// TIA Portal V16 program export: 4 tag tables, 2 data types, 7 data blocks, 42 code blocks (in call order from the OBs), 94 instance data blocks

VAR_GLOBAL   // PLC tag table "Default tag table"
   "Drive 1 Ready" AT %I0.0 : Bool;   // +MC-21K2:1 - Drive 1 Ready
   "Drive 2 Ready" AT %I0.1 : Bool;   // +MC-21K2:5 - Drive 2 Ready
   "Drive 3 Ready" AT %I0.2 : Bool;   // +MC-21K2:2 - Drive 3 Ready
   "Drive 4 Ready" AT %I0.3 : Bool;   // +MC-21K2:6 - Drive 4 Ready
   "Drive 5 Ready" AT %I0.4 : Bool;   // +MC-21K2:3 - Drive 5 Ready
   "Sensor Trechter" AT %I0.5 : Bool;   // +MC-21K2:7 - Sensor Trechter
   "Sensor Op Band" AT %I0.6 : Bool;   // +MC-21K2:4 Sensor Op Band
   "Sensor Wals (Option)" AT %I0.7 : Bool;   // +MC-21K2:8 - Sensor Wals (Option)
   "ESB Oke" AT %I1.0 : Bool;   // +MC-21K3:1 - ESB Oke
   "ESB Pressend" AT %I1.1 : Bool;   // +MC-21K3:5 - ESB Pressend
   "Reset Active" AT %I1.2 : Bool;   // +MC-21K3:2 - Reset Active
   "Noodsleutel(1)" AT %I1.3 : Bool;   // +MC-21K3:6 - NOODSLEUTEL
   "Alle uitgangen(1)" AT %I1.4 : Bool;   // +MC-21K3:3 - Alle uitgangen
   "Door 1 NC contact" AT %I1.5 : Bool;   // +MC-21K3:7 - Safety Doorswitch 1
   "Door 1 NO contact" AT %I1.6 : Bool;   // +MC-21K3:4 - Safety Doorswitch 1 Normaly open
   "Door 2 NC contact" AT %I1.7 : Bool;   // +MC-21K3:8 - Safety Doorswitch 2
   "Spare(5)" AT %I3.0 : Bool;
   "Spare(6)" AT %I3.1 : Bool;
   "Spare(10)" AT %I180.0 : Bool;   // Spare
   "Spare(11)" AT %I180.1 : Bool;   // Spare
   "Spare(12)" AT %I3.4 : Bool;   // Spare
   "Spare(13)" AT %I3.5 : Bool;   // Spare
   "Spare(14)" AT %I3.6 : Bool;   // Spare
   "Spare(15)" AT %I3.7 : Bool;   // Spare
   "Programma 1" AT %I2.0 : Bool;   // +MC-21K4:1 - Programma 1
   "Programma 2" AT %I2.1 : Bool;   // +MC-21K4:5 - Programma 2 (Option)
   "Programma 3" AT %I2.2 : Bool;   // +MC-21K4:2 - Programma 3
   Cleaning AT %I2.3 : Bool;   // +MC-21K4:6 - Cleaning
   "Start Machine" AT %I2.4 : Bool;   // +MC-21K4:3 - Start Machine
   "Stop Machine" AT %I2.5 : Bool;   // +MC-21K4:7 - Stop Machine
   "Spare(16)" AT %I2.6 : Bool;   // Spare
   Encoder_Z_Puls AT %I2.7 : Bool;   // Spare
   "Safety Relais" AT %Q0.0 : Bool;   // +MC-21K6:1 - Safety Relais
   "Bel Storing" AT %Q0.1 : Bool;   // +MC-21K6:5 - Bel Storing
   Spare AT %Q5.3 : Bool;   // Spare
   "Drive 1 RUN FWD" AT %Q1.0 : Bool;   // +MC-21K8:1 - Drive 1 RUN FWD
   "Drive 1 REV]" AT %Q1.1 : Bool;   // +MC-21K8:5 - Drive 1 REV
   "Drive 1 Speed 1" AT %Q1.2 : Bool;   // +MC-21K8:2 - Drive 1 Speed 1
   "Drive 1 Speed 2" AT %Q1.3 : Bool;   // +MC-21K8:6 - Drive 1 Speed 2
   "Spare(3)" AT %Q1.4 : Bool;   // Spare
   "Drive 2 RUN FWD" AT %Q1.5 : Bool;   // +MC-21K8:7 - Drive 2 RUN FWD
   "Drive 2 REV" AT %Q1.6 : Bool;   // +MC-21K8:4 - Drive 2 REV
   "Drive 2 Speed 1" AT %Q1.7 : Bool;   // +MC-21K8:8 - Drive 2 Speed 1
   "Drive 2 Speed 2" AT %Q2.0 : Bool;   // +MC-21K9:1 - Drive 2 Speed 2
   "Spare(4)" AT %Q2.1 : Bool;   // Spare
   "Drive 3 RUN FWD" AT %Q2.2 : Bool;   // +MC-21K9:2 - Drive 3 RUN FWD
   "Drive 3 REV" AT %Q2.3 : Bool;   // +MC-21K9:6 - Drive 3 REV
   "Drive 3 Speed 1" AT %Q2.4 : Bool;   // +MC-21K9:3 - Drive 3 Speed 1
   "Drive 3 Speed 2" AT %Q2.5 : Bool;   // +MC-21K9:7 - Drive 3 Speed 2
   "Spare(21)" AT %Q2.6 : Bool;   // Spare
   "Drive 4 RUN FWD" AT %Q2.7 : Bool;   // +MC-21K9:8 - Drive 4 RUN FWD
   "Drive 4 REV" AT %Q3.0 : Bool;   // +MC-21K10:1 - Drive 4 REV
   "Drive 4 Speed 1" AT %Q3.1 : Bool;   // +MC-21K10:5 - Drive 4 Speed 1
   "Drive 4 Speed 2" AT %Q3.2 : Bool;   // +MC-21K10:2 - Drive 4 Speed 2
   "Spare(22)" AT %Q3.3 : Bool;   // Spare
   "Drive 5 RUN FWD" AT %Q3.4 : Bool;   // +MC-21K10:3 - Drive 5 RUN FWD
   "Drive 5 REV" AT %Q3.5 : Bool;   // +MC-21K10:7 - Drive 5 REV
   "Drive 5 Speed 1" AT %Q3.6 : Bool;   // +MC-21K10:4 - Drive 5 Speed 1
   "Drive 5 Speed 2" AT %Q3.7 : Bool;   // +MC-21K10:8 - Drive 5 Speed 2
   "Spare(23)" AT %Q4.0 : Bool;   // Spare
   "LED Programma 1" AT %Q4.1 : Bool;   // +MC-21K11:5 - LED Programma 1
   "LED Programma 2" AT %Q4.2 : Bool;   // +MC-21K11:2 - LED Programma 2
   "LED Programma 3" AT %Q4.3 : Bool;   // +MC-21K11:6 - LED Programma 3
   "LED E-STOP" AT %Q0.2 : Bool;   // +MC-21K6:2- LED E-STOP
   "LED RUN" AT %Q4.5 : Bool;   // +MC-21K11:7 - LED RUN
   "Valve 1" AT %Q4.6 : Bool;   // +MC-21K11:4 - Valve 1
   "Valve 2" AT %Q4.7 : Bool;   // +MC-21K11:8 - Valve 2
   "Valve 3" AT %Q5.0 : Bool;   // +MC-21K12:1 - Valve 3
   "Valve 4" AT %Q5.1 : Bool;   // +MC-21K12:5 - Valve 4
   "Valve 5" AT %Q5.2 : Bool;   // +MC-21K12:2 - Valve 5
   Nootstopper AT %Q6.0 : Bool;   // Spare
   "Spare(2)" AT %Q6.1 : Bool;   // Spare
   "Spare(18)" AT %Q6.2 : Bool;   // Spare
   "Spare(19)" AT %Q6.3 : Bool;   // Spare
   "Spare(20)" AT %Q4.4 : Bool;   // Spare
   "Drive 1 Rapid Stop" AT %Q0.3 : Bool;   // +MC-21K6:6 - Drive 1 Rapid Stop
   "Drive 2 Rapid Stop" AT %Q0.4 : Bool;   // +MC-21K6:3 - Drive 2 Rapid Stop
   "Drive 3 Rapid Stop" AT %Q0.5 : Bool;   // +MC-21K6:7 - Drive 3 Rapid Stop
   "Drive 4 Rapid Stop" AT %Q0.6 : Bool;   // +MC-21K6:4 - Drive 4 Rapid Stop
   "Drive 5 Rapid Stop" AT %Q0.7 : Bool;   // +MC-21K6:8 - Drive 5 Rapid Stop
   "Systeem RUN" AT %M0.0 : Bool;   // Systeem RUN
   Tag_1 AT %M0.1 : Bool;
   Tag_2 AT %M0.2 : Bool;
   Tag_3 AT %M0.3 : Bool;
   Tag_4 AT %M0.4 : Bool;
   "Safety Feedback" AT %M0.6 : Bool;
   Tag_5 AT %M0.7 : Bool;
   Tag_6 AT %M1.0 : Bool;
   "ONC Drive 1 RUN FWD" AT %M10.0 : Bool;
   "ONC Drive 2 RUN FWD" AT %M10.1 : Bool;
   "ONC Drive 3 RUN FWD" AT %M10.2 : Bool;
   "ONC Drive 4 RUN FWD" AT %M10.3 : Bool;
   "ONC Drive 5 RUN FWD" AT %M10.4 : Bool;
   "ONC Drive 1 RUN FWD and Speed 1" AT %M10.5 : Bool;
   "ONC Drive 2 RUN FWD and Speed 1" AT %M10.6 : Bool;
   "ONC Drive 3 RUN FWD and Speed 1" AT %M10.7 : Bool;
   "ONC Drive 4 RUN FWD and Speed 1" AT %M11.0 : Bool;
   "ONC Drive 5 RUN FWD and Speed 1" AT %M11.1 : Bool;
   "ONC Drive 1 RUN FWD and Speed 2" AT %M11.2 : Bool;
   "ONC Drive 2 RUN FWD and Speed 2" AT %M11.3 : Bool;
   "ONC Drive 3 RUN FWD and Speed 2" AT %M11.4 : Bool;
   "ONC Drive 4 RUN FWD and Speed 2" AT %M11.5 : Bool;
   "ONC Drive 5 RUN FWD and Speed 2" AT %M11.6 : Bool;
   Startknop_Scherm AT %M15.0 : Bool;
   Stopknop_Scherm AT %M15.1 : Bool;
   Tag_7 AT %M110.1 : Bool;
   Reset_scherm AT %M15.2 : Bool;
   Sensor_op_band_memory AT %M15.3 : Bool;
   "System RUN_1" AT %M20.0 : Bool;
   ResetDelay AT %M20.1 : Bool;
   SensorWalsMemory AT %M20.2 : Bool;
   Timer_Memory AT %M20.3 : Bool;
   StopAll AT %M20.4 : Bool;
   Tag_8 AT %M100.3 : Bool;
   Tag_9 AT %M100.4 : Bool;
   Tag_10 AT %M0.5 : Bool;
   Tag_11 AT %M150.0 : Bool;
   Tag_12 AT %M101.1 : Bool;
   Tag_13 AT %T1 : Timer;
   Tag_14 AT %M300.0 : Bool;
   Tag_15 AT %M260.0 : Bool;
   Tag_16 AT %M300.1 : Bool;
   Tag_17 AT %M501.0 : Bool;
   Tag_18 AT %M500.1 : Bool;
   Tag_19 AT %M160.0 : Bool;
   Tag_20 AT %M150.5 : Bool;
   Tag_21 AT %QD256 : DWord;
   Tag_22 AT %QW260 : Word;
   Tag_23 AT %ID256 : DWord;
   Tag_24 AT %ID260 : DWord;
   Tag_25 AT %ID464 : DWord;
   Tag_26 AT %ID471 : DWord;
   Tag_27 AT %QW471 : Word;
   Tag_28 AT %QD464 : DWord;
   Tag_30 AT %IW205 : Int;
   SystemTime AT %MD2 : Time;
   Tag_31 AT %M5.0 : Bool;
   Lamp_Green AT %Q7.0 : Bool;
   Lamp_Blue AT %Q7.1 : Bool;
   Lamp_Yellow AT %Q7.2 : Bool;
   Lamp_Red AT %Q7.3 : Bool;
   Lamp_Buzzer AT %Q7.4 : Bool;
   PulseTimer AT %T0 : Timer;
   Zpuls_Encoder_Band_Set AT %M1.1 : Bool;
   Drive_1_RefRun AT %M1.2 : Bool;
   Tag_32 AT %QD110 : DWord;
   Tag_33 AT %QD111 : DWord;
   Tag_34 AT %QD112 : DWord;
   Tag_35 AT %QD113 : DWord;
   Tag_36 AT %QD114 : DWord;
   Tag_37 AT %QD115 : DWord;
   Tag_38 AT %QD116 : DWord;
   Tag_39 AT %QD117 : DWord;
   Tag_40 AT %QB110 : Byte;
   Tag_41 AT %QB111 : Byte;
   Tag_42 AT %QB112 : Byte;
   Tag_43 AT %QB113 : Byte;
   Tag_44 AT %IB110 : Byte;
   Tag_45 AT %IB111 : Byte;
   Tag_46 AT %IB112 : Byte;
   Tag_47 AT %IB113 : Byte;
   Tag_48 AT %IB114 : Byte;
   Tag_49 AT %IB115 : Byte;
   Tag_50 AT %IB116 : Byte;
   Tag_51 AT %IB117 : Byte;
   Tag_52 AT %QD260 : DWord;
   Tag_53 AT %QB114 : Byte;
   Tag_54 AT %QB115 : Byte;
   Tag_55 AT %QB116 : Byte;
   Tag_56 AT %QB117 : Byte;
   Tag_57 AT %QW256 : Word;
   Tag_58 AT %QW258 : Word;
   Tag_59 AT %IW256 : Word;
   Tag_60 AT %IW258 : Word;
   Tag_61 AT %QW112 : Word;
   "Blow Off Timed" AT %M1.3 : Bool;
   Stop_valve_6 AT %M1.4 : Bool;
   Valve_6_Manual AT %M1.5 : Bool;
   Valve_6_Auto AT %M1.6 : Bool;
END_VAR

VAR_GLOBAL   // PLC tag table "PositionControl"
   Counter1_IW100 AT %IW100 : Int;
   Counter2_IW102 AT %IW102 : Int;
   "Manual Jog Fwd" AT %M137.0 : Bool;
   "Manual Jog Rev" AT %M137.1 : Bool;
   ReferenceSwitchAxis3 AT %I3.0 : Bool;
   EncoderBand_Alive AT %IW110 : Int;
   EncoderBand_RawCounter AT %ID112 : DInt;
   EncoderBand_FineCounter AT %IW113 : Int;
   Zpuls_Encoder_Band AT %I110.3 : Bool;
   Enc1 AT %ID110 : DInt;
   Enc2 AT %ID111 : DInt;
   Enc3 AT %ID113 : DInt;
   "Zpuls_Encoder_Band(1)" AT %I113.3 : Bool;
   "Enc3(1)" AT %ID114 : DInt;
   "Enc3(2)" AT %ID115 : DInt;
   "Enc3(3)" AT %ID116 : DInt;
   "Enc3(4)" AT %ID117 : DInt;
   "Enc3(5)" AT %ID118 : DInt;
   "Enc3(6)" AT %IW112 : Int;
   Enable AT %QW110 : Word;
   MovePos2 AT %M222.0 : Bool;
   ActivateProductBufferV3 AT %M222.1 : Bool;
END_VAR

VAR_GLOBAL   // PLC tag table "Secund. Tags"
   Aanvoerband_Tag1 AT %M100.0 : Bool;
   Aanvoerband_Tag2 AT %M100.1 : Bool;
   Trechter_Bijvullen_Haltveroorzaker AT %M100.2 : Bool;
   Safety_Automatic AT %M100.5 : Bool;
   Safety_Override AT %M100.6 : Bool;
   RUN_Automatic AT %M100.7 : Bool;
   RUN_Manual AT %M101.0 : Bool;
   Invert_Trechter_Sensor AT %M101.2 : Bool;
   WalsSensorMemory AT %M101.3 : Bool;
   Disable_Module AT %M101.4 : Bool;
   Sensor_Trechter_Delayed AT %M101.5 : Bool;
   Positive_Flank AT %M101.6 : Bool;
   ProductSensor_Flank AT %M101.7 : Bool;
   ProductSensor_Rug AT %M102.0 : Bool;
   SensorRug AT %M102.1 : Bool;
   TimeCyclusEnd AT %M102.2 : Bool;
   CounterReset AT %M102.3 : Bool;
   StartTimer AT %M102.4 : Bool;
   StopTimer AT %M102.5 : Bool;
   SaveTimervalue AT %M102.6 : Bool;
   ResetTotalProducts AT %M102.7 : Bool;
   MaintenanceNeeded AT %M103.0 : Bool;
   RetainValues AT %M112.0 : Bool;
   "Retain_1_DontTouch!" AT %M112.1 : Bool;
   Safety_Doors AT %M112.2 : Bool;
   Overname_Linked_Drive1 AT %M112.3 : Bool;
   Drive_RefuseLinkingDrive1 AT %M112.4 : Bool;
   Drive_4_Speed1_Link AT %M112.5 : Bool;
   Drive_4_Speed1_Unlink AT %M112.6 : Bool;
   SafetyOK AT %M112.7 : Bool;
   Valve2_Pulse AT %M113.0 : Bool;
   TurnOffDrive2 AT %M113.1 : Bool;
   TurnOffDrive4 AT %M113.2 : Bool;
   TurnOff_InfeedTimeout AT %M113.3 : Bool;
END_VAR

VAR_GLOBAL   // PLC tag table "Tag table_1"
END_VAR

TYPE "ProductEntry"
// stored: IsFailsafeCompliant false
   STRUCT
      StartTime : Time := T#0ms;
      Active : Bool;
   END_STRUCT;
END_TYPE

TYPE "ProductTrack"
// stored: IsFailsafeCompliant false
   STRUCT
      StartPosition : DInt;
      Active : Bool;
   END_STRUCT;
END_TYPE

DATA_BLOCK "DB1"   // DB93
VERSION : 0.1
// stored: AutoNumber true, IsOnlyStoredInLoadMemory false, IsWriteProtectedInAS false
   VAR RETAIN
      DBB0 : DWord;
      DBB15 : DWord;
      DBB14 : DWord;
      DBB13 : DWord;
      DBB12 : DWord;
      DBB11 : DWord;
      DBB10 : DWord;
      DBB9 : DWord;
      DBB8 : DWord;
      DBB7 : DWord;
      DBB6 : DWord;
      DBB5 : DWord;
      DBB4 : DWord;
      DBB3 : DWord;
      DBB2 : DWord;
      DBB1 : DWord;
      DBD4 : DWord;
      DBD0 : DWord;
      "DBX4.0" : Bool;
   END_VAR
BEGIN
END_DATA_BLOCK

DATA_BLOCK "DB_EncoderBand"   // DB95
VERSION : 0.1
// stored: AutoNumber false, IsOnlyStoredInLoadMemory false, IsWriteProtectedInAS false
   VAR RETAIN
      ControlWord1 : DInt;
      ControlWord2 : DInt;
      FeedbackWord1 : DInt;
      FeedbackWord2 : DInt;
      EnableGate : Bool;
      ControlWord : Word;
      EncoderValue : DInt;
   END_VAR
BEGIN
END_DATA_BLOCK

DATA_BLOCK "Datablock_Encoder"   // DB96
VERSION : 0.1
// stored: AutoNumber true, IsOnlyStoredInLoadMemory false, IsWriteProtectedInAS false
BEGIN
END_DATA_BLOCK

DATA_BLOCK "PLCMemory"   // DB15
VERSION : 0.1
// stored: AutoNumber true, IsOnlyStoredInLoadMemory false, IsWriteProtectedInAS false
   VAR RETAIN
      Homing_Sensor_Wals_Offset_Test : Time := T#1S_200MS;   // Offset of homing position sensor wals
      Wals_Delay_Offset : Time := T#400MS;   // Offset of Wals on delay
      Safety_Delay : Time := T#5MS;   // Delay of safety high
      WalsCheck_Time : Time := T#5S;   // Time offset when wals slipping message is displayed
      ProductCheck_Time : Time := T#15S;   // Time offset when aanvoer not in position message is displayed
      ProductIntervalTime : Time := T#10s;   // Counts the time between 2 products
      ProductIntervalTime_1 : Time;   // Depends on ProductIntervalTimer
      ProductIntervalTime_2 : Time;   // Depends on ProductIntervalTimer_1
      TD_Products_Counter : Int;   // Counts the total amount of products with the Sensor Band
      UsernameMemory : String := 'Key';
      PasswordMemory : String := 'Key123';
      SpeedSettingsTakeover : Bool := True;   // Makes the speed of Overname the same as speed Drive 1
      SpeedSettingOvername : Bool;   // Parameter of setting the speed for Drive 4 (Overname)
      SpeedSettingBand : Bool;   // Parameter of setting the speed for Drive 1 (Band)
      TimingSettingOvername : Bool := True;   // Makes the timing of Overname the same as speed Drive 1
      EncoderPosition : Real;   // Real Value of Encoder Axis 3 (Wals)
      StepSize : Real := 0.0;   // Pulsfactor of Encoder Axis 3
      Desired_Encoder_Position : Real;
      Tolerance : Real := 0.0;
      "Encoder PulsOffset" : Time := T#3MS;
      Axis3_Ref_Pos : Real := 85.0;   // Refention position of Axis 3 without tolerance
      Reference_Position_Axis3 : Real;   // Refention position of Axis 3 with calculated tolerance
      ProductCount : Int;
      Axis3_ControlMode : Bool := true;
      Axis1_ControlMode : Bool := true;
      ProductsToProduce : Int;
      SystemTime : Time;
      Disable_Modules : Struct
         Disable_Band : Bool;
         Disable_Trilgoten : Bool;
         Disable_AanvoerWals : Bool;
         Disable_Aandruk1 : Bool;
         Disable_Aandruk2 : Bool;
         Disable_Aandruk3 : Bool;
         Disable_Blaaspuls : Bool;
         Disable_Retourband : Bool;
         Disable_Afsluiter : Bool;
         Disable_Nootstopper : Bool;
      END_STRUCT;
      Offset_Timers : Struct
         Trilgoten_Start_Offset : Time := T#10MS;   // Delay offset of start trilgoten
         Trilgoten_Stop_Offset : Time := T#10MS;   // Delay offset of stop trilgoten
         Aanvoer_Start_Offset : Time := T#10MS;   // Delay offset of start aanvoer
         Magazijn_Sensor_Delay : Time := T#15S;   // Delay on magazijn sensor.
         Aanvoer_Stop_Offset : Time := T#10MS;   // Delay offset of stop aanvoer
         Overname_Start_Offset : Time := T#5MS;   // Delay offset of start Overname
         Overname_Stop_Offset : Time := T#5MS;   // Delay offset of stop Overname
         Retourband_Start_Offset : Time := T#5ms;
         Retourband_Stop_Offset : Time := T#5ms;
         BlowOff_CycleTime : Time := T#500ms;
         Blow_Off_PulseTime : Time := T#500ms;
      END_STRUCT;
      ProductBuffer : Struct
         DelayTime : Time := T#7s;
         ProductsCount : Int;
         MoveTrigger : Bool;
         MoveFeedback : Bool;
         RestFeedback : Bool;
         InsertIndex : Int;
      END_STRUCT;
      ProductBufferBehindWals : Struct
         DelayTime : Time := T#1s_890MS;
         Product_Count : Int;
      END_STRUCT;
      ProductBufferNutStopper : Struct
         ProductCount : Int;
         TimeOpenNutstopper_PT : Time := T#200MS;
         TimeOpenNutstopper_ET : Time;
      END_STRUCT;
      ProductBuffer_1 : Struct
         DelayTime : Time := T#7s;
         ProductsCount : Int;
         MoveTrigger : Bool;
         MoveFeedback : Bool;
         RestFeedback : Bool;
         InsertIndex : Int;
      END_STRUCT;
      TriggerDistanceBand : DInt := 418000;
      TriggerDistanceAandruk : DInt := 500000;
      TriggerDistanceNutStopper : DInt := 459000;
      InfeedTimeOutPT : Time := T#2S;
      "Blow Off Timer on" : Time := T#2S;
      ResetManual : Bool;
      StartDevTestingInfeedSensor : Bool;
      SimulateSensor : Bool;
      PulsTimeBlowOff : Time := T#650ms;
      BlowOffPulse : Bool;
      OutputUserText : Struct
         Axis1 : Struct
            "User1.Text" : String := '(300) Manual Jogging';
            "User2.Text" : String := '(50) Automatic Production';
            "User3.Text" : String := '(1) Reference Run';
            "User4.Text" : String;
            CurrentUserText : String;
         END_STRUCT;
         Axis2 : Struct
            "User1.Text" : String := '(300) Manual Jogging';
            "User2.Text" : String := '(50) Automatic Production';
            "User3.Text" : String;
            "User4.Text" : String;
            CurrentUserText : String;
         END_STRUCT;
         Axis3 : Struct
            "User1.Text" : String := '(300) Manual Jogging Fwd';
            "User2.Text" : String := '(300) Manual Jogging Rev';
            "User3.Text" : String := '(50) Automatic Servomanager';
            "User4.Text" : String := '(1) Reference Run';
            CurrentUserText : String;
         END_STRUCT;
         Axis4 : Struct
            "User1.Text" : String := '(300) Manual Jogging';
            "User2.Text" : String := '(50) Automatic Production';
            "User3.Text" : String;
            "User4.Text" : String;
            CurrentUserText : String;
         END_STRUCT;
         Axis5 : Struct
            "User1.Text" : String := '(300) Manual Jogging';
            "User2.Text" : String := '(50) Automatic Production';
            "User3.Text" : String;
            "User4.Text" : String;
            CurrentUserText : String;
         END_STRUCT;
      END_STRUCT;
      Modules : Struct
         Valve_6 : "ModuleOutput";
         Valve_1 { S7_SetPoint := 'True'} : "ModuleOutput";
         Valve_3 { S7_SetPoint := 'True'} : "ModuleOutput";
         Valve_4 { S7_SetPoint := 'True'} : "ModuleOutput";
         Valve_5 { S7_SetPoint := 'True'} : "ModuleOutput";
      END_STRUCT;
   END_VAR
BEGIN
END_DATA_BLOCK

DATA_BLOCK "DB_SystemTimeCounter"   // DB68
VERSION : 0.1
// stored: AutoNumber true, IsOnlyStoredInLoadMemory false, IsWriteProtectedInAS false
   VAR RETAIN
      SystemTime : Time;
   END_VAR
BEGIN
END_DATA_BLOCK

DATA_BLOCK "Alarms"   // DB24
VERSION : 0.1
// stored: AutoNumber true, IsOnlyStoredInLoadMemory false, IsWriteProtectedInAS false
   VAR
      AlarmStruct : Struct
         Alarm_Product_Not_Position : Bool;
         Alarm_Axis_Not_Position : Bool;
         Alarm_Drive1 : Bool;
         Alarm_Drive2 : Bool;
         Alarm_Drive3 : Bool;
         Alarm_Drive4 : Bool;
         Alarm_Drive5 : Bool;
         "Alarm_To_Many_Products_Reset_Counter!" : Bool;
      END_STRUCT;
      AlarmsWord : Word;
      HMI_Alarm_Drive1 : Word;
      HMI_Alarm_Drive2 : Word;
      HMI_Alarm_Drive3 : Word;
      HMI_Alarm_Drive4 : Word;
      HMI_Alarm_Drive5 : Word;
   END_VAR
BEGIN
END_DATA_BLOCK

DATA_BLOCK "PositionManagement"   // DB51
VERSION : 0.1
// stored: AutoNumber true, IsOnlyStoredInLoadMemory false, IsWriteProtectedInAS false
   VAR RETAIN
      Data : Struct   // Data
         CntPlsPrev : DInt := 0;   // Flowpulsen vorige scan
         CntPlsDiff : DInt := 0;   // Flowpulsen verschil
         CntPlsAct : DInt := 0;   // Flowpulsen actueel
         DosActueel : Real := 0.0;   // Dosering actueel (not used)
         Actual_Axis3_Position : Real;   // Actual Position of Axis 3 stored in this datablock
         Actual_Axis1_Position : Real;
      END_STRUCT;
      "Axis 3" : Struct
         Values : Struct
            AxisName : String := 'Drive 3 - Wals';
            "Reference Position" : Int := 0;
            "Set Position" : Real := -50.0;
            "Rest Position" : Real := -25.0;
            Acceleration : Real := 0.0;
            Deacceleration : Real;
            "Axis Correction" : Real := 1.0E-06;
            "Position Offset" : Real := 35.0;
            Pulsfactor : Real := 0.82;
            Axis_Speed : Int := 0;
            ModuloFactor : Real := 360.0;
         END_STRUCT;
         Commands : Struct
            "Go To Rest" : Bool;
            "Start Ref Run" : Bool;
            "Take Over Pos" : Bool;
            "Go To Position" : Bool;
            "Jog Fwd" : Bool;
            "Jog Rev" : Bool;
            Axis_Brake : Bool;
            MasterWord : String;
            "Master Callback" : String;
         END_STRUCT;
         Messages : Struct
            "Axis Busy" : Bool;
            "Error Executing Command" : Bool;
            "Axis On Rest" : Bool;
            "Axis On Position" : Bool;
            "Drive State (Option)" : String;
            "Slip State" : String;
            AxisHasReference : Bool;
         END_STRUCT;
      END_STRUCT;
      Demo_Pos : Struct
         Desired_Pos : Real;
         Start : Bool;
         SetRefRunActive : Bool;
         RequestMove1 : Bool;
         RequestMove2 : Bool;
         PositionMove2 : Real := -50.0;
         PositionMove1 : Real := -250.0;
         Pos2Done : Bool;
         BrakeOnPos1 : Bool;
         BrakeOnPos2 : Bool;
         ManualSensorOverride : Bool;
      END_STRUCT;
      Axis_1 : Struct
         Values : Struct
            AxisName : String := 'Drive 1 - Infeed';
            "Reference Position" : Int := 0;
            "Set Position" : Real := 0.0;
            "Rest Position" : Real := 0.0;
            Acceleration : Real := 0.0;
            Deacceleration : Real;
            "Axis Correction" : Real := 1.0E-06;
            "Position Offset" : Real := 0.001;
            Pulsfactor : Real := -0.359;
            Axis_Speed : Int := 0;
            LimitEncValue : DInt := 0;
         END_STRUCT;
         Commands : Struct
            "Go To Rest" : Bool;
            "Start Ref Run" : Bool;
            "Take Over Pos" : Bool;
            "Go To Position" : Bool;
            "Jog Fwd" : Bool;
            "Jog Rev" : Bool;
            Axis_Brake : Bool;
            ReferenceSwitch : Bool;
            MasterWord : String;
            "Master Callback" : String;
         END_STRUCT;
         Messages : Struct
            "Axis Busy" : Bool;
            "Error Executing Command" : Bool;
            "Axis On Rest" : Bool;
            "Axis On Position" : Bool;
            "Drive State (Option)" : String;
            "Slip State" : String;
            AxisHasReferenceDelayed : Bool;
            AxisHasReference : Bool;
            SetAxisHasRefFromEnc : Bool;
            MaxOverflowValueDint : DInt := 16#8261A800;
         END_STRUCT;
      END_STRUCT;
   END_VAR
BEGIN
END_DATA_BLOCK

ORGANIZATION_BLOCK "OB1"   // OB1, LAD, ProgramCycle
TITLE = MAIN Program - Sweep
VERSION : 0.1
// MAIN Program Block (Release)
// stored: IsIECCheckEnabled false
   VAR_TEMP
      Temp_0 : Byte;
      Temp_1 : Byte;
      Temp_2 : Byte;
      Temp_3 : Byte;
      Temp_4 : Byte;
      Temp_5 : Byte;
      Temp_6 : Int;
      Temp_7 : Int;
      Temp_8 : Int;
      Temp_9 : Date_And_Time;
      Temp_10 : DWord;
      EncoderDirection : Bool;
      HomingActive : Bool;
      EncError : Bool;
      SafetyActive : Bool;
      "Spare Drive 6" : Bool;
      "Spare Drive 7" : Bool;
      "Spare Drive 8" : Bool;
      "Spare Drive 9" : Bool;
      "Spare Drive 10" : Bool;
      SAFE_OK_Signal : Bool;
      Raw_Position : Real;
      Encoder : Int;
      Gate : Bool;
      GATESTP : Bool;
      OTERRA : Bool;
      Direct : Bool;
      Prepar : Bool;
      CMPV1 : Bool;
      CMPV2 : Bool;
      RESSYNC : Bool;
      RESZERO : Bool;
      OTERR : Bool;
      UnscPos : Int;
      Sc_Pos : Int;
      ActEncPos : Real;
      Start_ReferenceRun : Bool;
      ReferenceSwitch_Input : Bool;
      "Reference Position" : Real;
      "Jog FWD" : Bool;
      "Jog REV" : Bool;
      RefSwitchTemp : Bool;
      RefPosDint : DInt;
      RefPosInt : Real;
      Start_Movement : Bool;
      ClockTime : Int;
      LT_Time : Date_And_Time;
      Summer : Bool;
      SystemStartUp : Bool;
      StartupLow : Bool;
      ManualSensorOverride : Bool;
      Axis1_ScaledPosition : Real;
      Axis1_ActualEncPosition : Real;
      ActivateProductBufferV2 : Bool;
      ActivateProductBufferV3 : Bool;
      SetZPulse : Bool;
      Enc2_AboveZero : DInt;
      MinValue : DInt;
      EncBelowZero : Bool;
      SafeEncValue : Real;
      Enc2_Real : Real;
      ScPos : Real;
      UseOldDriveManager : Bool;
      NotUsed : Bool;
      Door2 : Bool;
      Resettt : Bool;
      BlkMovReturn : Int;
      BlkMovReturn2 : Int;
      ServoAxis3RefRun : Bool;
   END_VAR
   VAR_TEMP   // added for the SCL form of the ladder/FBD networks
      _w1 : Bool;
   END_VAR
BEGIN

REGION Network 1: System Startup
   // Network for detecting System Start-up.
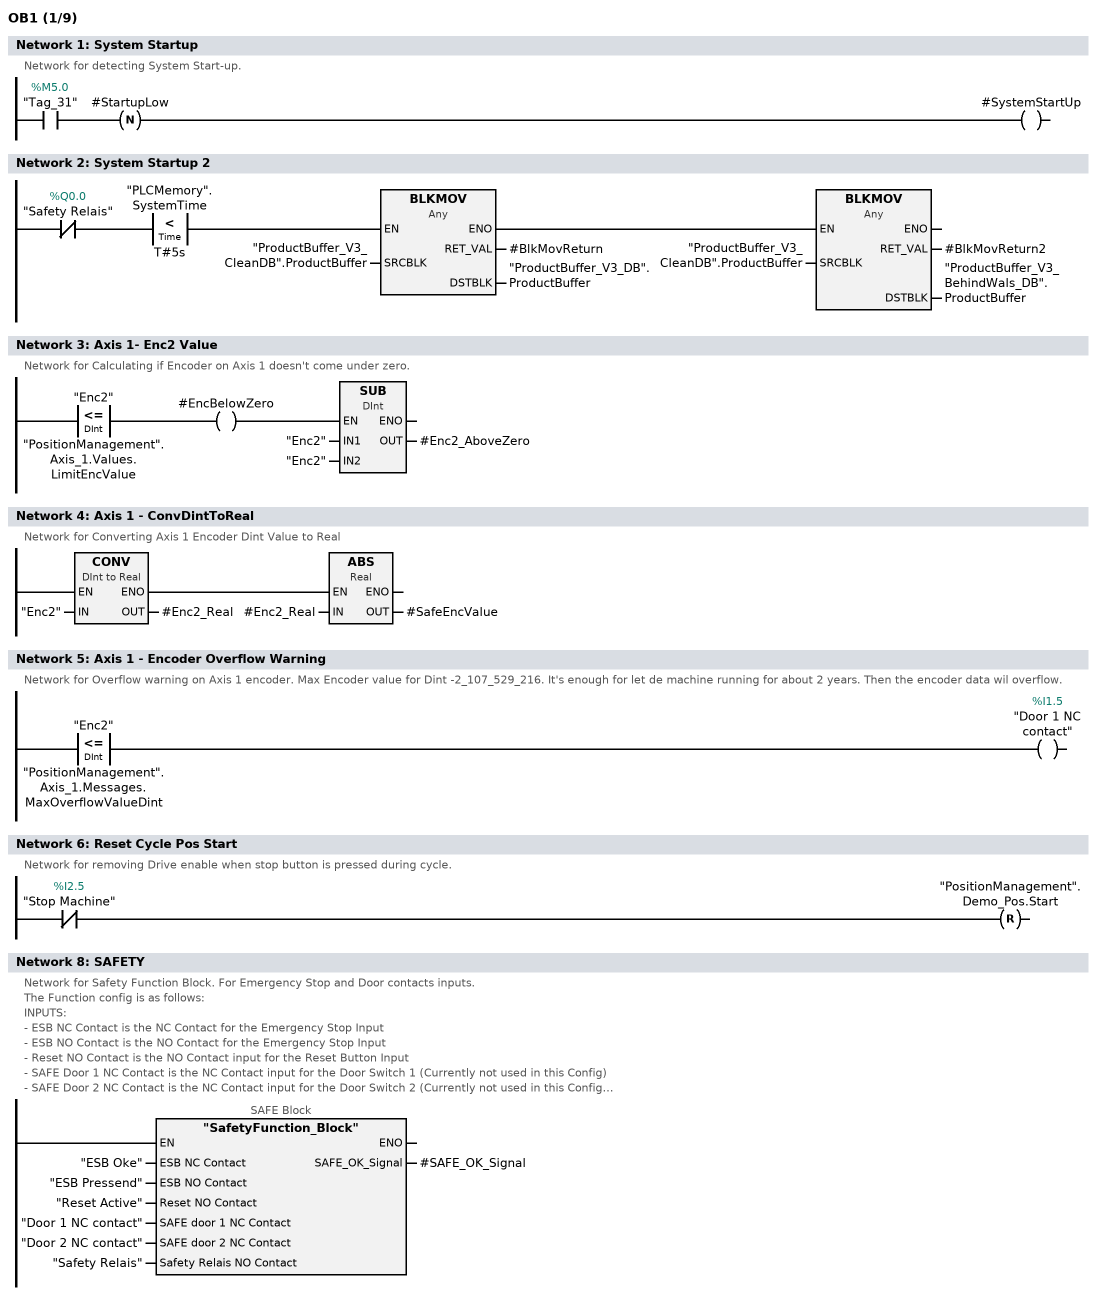
   RUNG wire#powerrail
      Contact( "Tag_31" )
      N_Trig( #StartupLow )
      Coil( #SystemStartUp )
   END_RUNG
   // the same network as SCL:
   #_w1 := NOT "Tag_31" AND #StartupLow;   // falling edge
   #StartupLow := "Tag_31";
   #SystemStartUp := #_w1;
END_REGION

REGION Network 2: System Startup 2
   RUNG wire#powerrail
      I_Contact( "Safety Relais" )
      { S7_Templates := "SrcType := Time" } LT_Contact(in1 := "PLCMemory".SystemTime, in2 := T#5s)
      { S7_Templates := "blk_type := Any" } BLKMOV(SRCBLK := "ProductBuffer_V3_CleanDB".ProductBuffer, RET_VAL => #BlkMovReturn, DSTBLK => "ProductBuffer_V3_DB".ProductBuffer)
      { S7_Templates := "blk_type := Any" } BLKMOV(SRCBLK := "ProductBuffer_V3_CleanDB".ProductBuffer, RET_VAL => #BlkMovReturn2, DSTBLK => "ProductBuffer_V3_BehindWals_DB".ProductBuffer)
   END_RUNG
   // the same network as SCL:
   #BlkMovReturn := BLKMOV(EN := NOT "Safety Relais" AND ("PLCMemory".SystemTime < T#5s),
                           SRCBLK := "ProductBuffer_V3_CleanDB".ProductBuffer,
                           DSTBLK => "ProductBuffer_V3_DB".ProductBuffer,
                           ENO => #_w1);
   IF #_w1 THEN
       #BlkMovReturn2 := BLKMOV(SRCBLK := "ProductBuffer_V3_CleanDB".ProductBuffer,
                               DSTBLK => "ProductBuffer_V3_BehindWals_DB".ProductBuffer);
   END_IF;
END_REGION

REGION Network 3: Axis 1- Enc2 Value
   // Network for Calculating if Encoder on Axis 1 doesn't come under zero.
   RUNG wire#powerrail
      { S7_Templates := "SrcType := DInt" } LE_Contact(in1 := "Enc2", in2 := "PositionManagement".Axis_1.Values.LimitEncValue)
      Coil( #EncBelowZero )
      { S7_Templates := "SrcType := DInt"; S7_GenerateENO := "TRUE" } Sub(in1 := "Enc2", in2 := "Enc2", out => #Enc2_AboveZero)
   END_RUNG
   // the same network as SCL:
   #EncBelowZero := "Enc2" <= "PositionManagement".Axis_1.Values.LimitEncValue;
   IF #EncBelowZero THEN #Enc2_AboveZero := "Enc2" - "Enc2"; END_IF;
END_REGION

REGION Network 4: Axis 1 - ConvDintToReal
   // Network for Converting Axis 1 Encoder Dint Value to Real
   RUNG wire#powerrail
      { S7_Templates := "[SrcType := DInt, DestType := Real]"; S7_GenerateENO := "TRUE" } Convert(in := "Enc2", out => #Enc2_Real)
      { S7_Templates := "SrcType := Real"; S7_GenerateENO := "TRUE" } Abs(in := #Enc2_Real, out => #SafeEncValue)
   END_RUNG
   // the same network as SCL:
   // ENO of a box is taken as its EN; it also drops when the box reports an error
   #Enc2_Real := DINT_TO_REAL("Enc2");
   #SafeEncValue := ABS(#Enc2_Real);
END_REGION

REGION Network 5: Axis 1 - Encoder Overflow Warning
   // Network for Overflow warning on Axis 1 encoder. Max Encoder value for Dint -2_107_529_216. It's enough for let de machine running for about 2 years. Then the encoder data wil overflow.
   RUNG wire#powerrail
      { S7_Templates := "SrcType := DInt" } LE_Contact(in1 := "Enc2", in2 := "PositionManagement".Axis_1.Messages.MaxOverflowValueDint)
      Coil( "Door 1 NC contact" )
   END_RUNG
   // the same network as SCL:
   "Door 1 NC contact" := "Enc2" <= "PositionManagement".Axis_1.Messages.MaxOverflowValueDint;
END_REGION

REGION Network 6: Reset Cycle Pos Start
   // Network for removing Drive enable when stop button is pressed during cycle.
   RUNG wire#powerrail
      I_Contact( "Stop Machine" )
      R_Coil( "PositionManagement".Demo_Pos.Start )
   END_RUNG
   // the same network as SCL:
   IF NOT "Stop Machine" THEN "PositionManagement".Demo_Pos.Start := FALSE; END_IF;
END_REGION

REGION Network 7: Retain Veriables (Not Used)
   // Spare Network Currently not used
END_REGION

REGION Network 8: SAFETY
   // Network for Safety Function Block. For Emergency Stop and Door contacts inputs.
   // The Function config is as follows:
   // 
   // INPUTS:
   // - ESB NC Contact is the NC Contact for the Emergency Stop Input
   // - ESB NO Contact is the NO Contact for the Emergency Stop Input
   // - Reset NO Contact is the NO Contact input for the Reset Button Input
   // - SAFE Door 1 NC Contact is the NC Contact input for the Door Switch 1 (Currently not used in this Config)
   // - SAFE Door 2 NC Contact is the NC Contact input for the Door Switch 2 (Currently not used in this Config)
   // - Safety Relais NO Contact is the NO Contact Input for feedback whenether the Safety Relais is powered or not.
   // 
   // OUTPUTS:
   // - SAFE_OK_Signal is the output for the SAFE OK signal, it's HIGH when all safety inputs are HIGH, en when Reset is given.
   RUNG wire#powerrail
      "SafetyFunction_Block"("ESB NC Contact" := "ESB Oke", "ESB NO Contact" := "ESB Pressend", "Reset NO Contact" := "Reset Active", "SAFE door 1 NC Contact" := "Door 1 NC contact", "SAFE door 2 NC Contact" := "Door 2 NC contact", "Safety Relais NO Contact" := "Safety Relais", SAFE_OK_Signal => #SAFE_OK_Signal)   // SAFE Block
   END_RUNG
   // the same network as SCL:
   "SafetyFunction_Block"("ESB NC Contact" := "ESB Oke",   // SAFE Block
                          "ESB NO Contact" := "ESB Pressend",
                          "Reset NO Contact" := "Reset Active",
                          "SAFE door 1 NC Contact" := "Door 1 NC contact",
                          "SAFE door 2 NC Contact" := "Door 2 NC contact",
                          "Safety Relais NO Contact" := "Safety Relais",
                          SAFE_OK_Signal => #SAFE_OK_Signal);
END_REGION

REGION Network 9: SAFE Signal
   // Network for internal SAFETY OK Confirmation
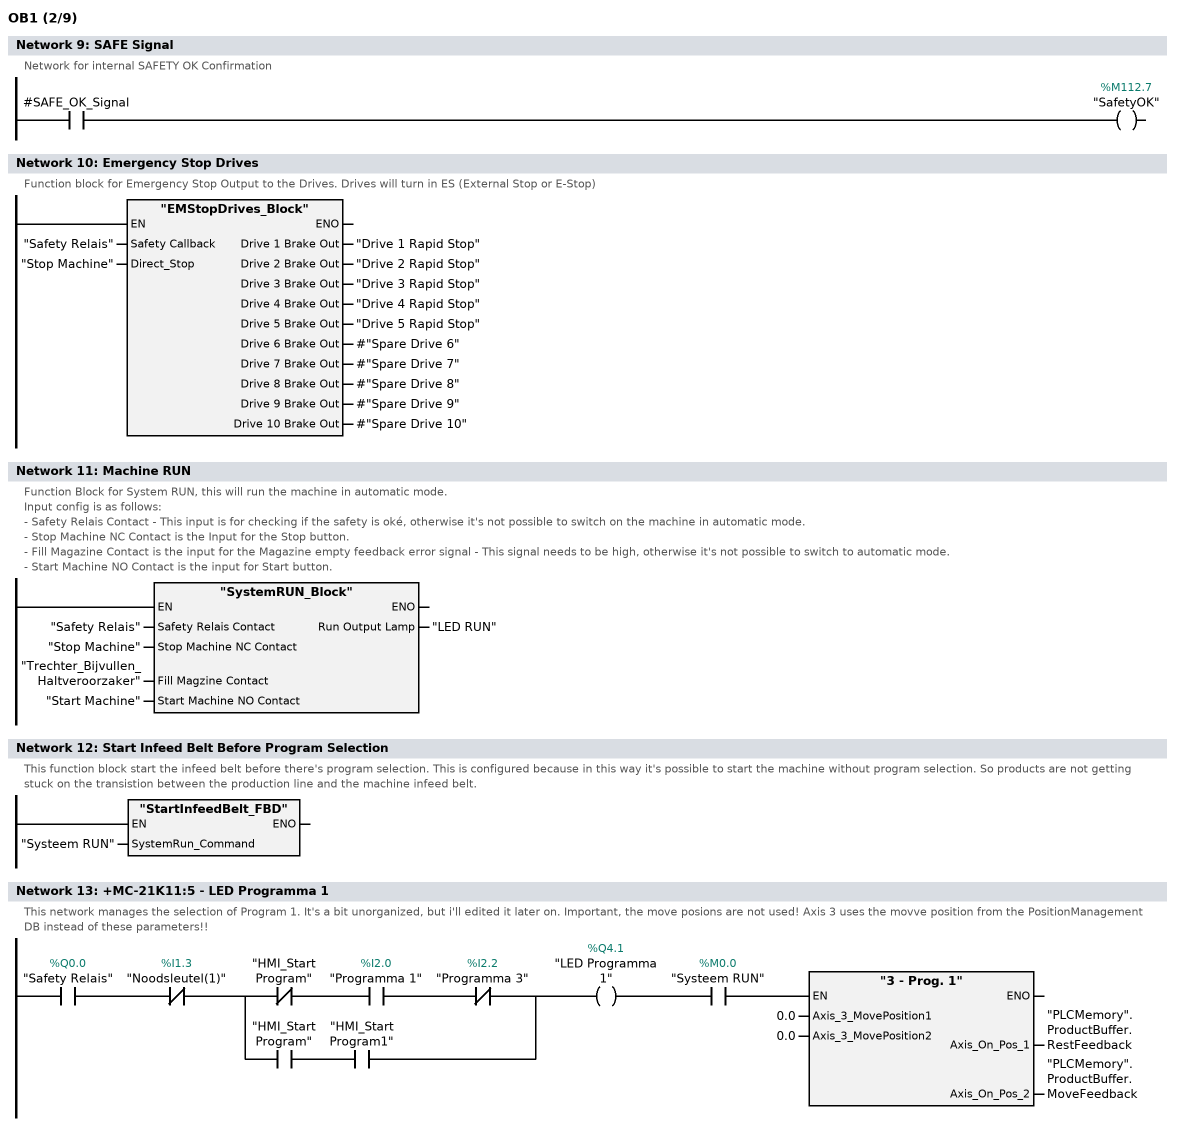
   RUNG wire#powerrail
      Contact( #SAFE_OK_Signal )
      Coil( "SafetyOK" )
   END_RUNG
   // the same network as SCL:
   "SafetyOK" := #SAFE_OK_Signal;
END_REGION

REGION Network 10: Emergency Stop Drives
   // Function block for Emergency Stop Output to the Drives. Drives will turn in ES (External Stop or E-Stop)
   RUNG wire#powerrail
      "EMStopDrives_Block"("Safety Callback" := "Safety Relais", Direct_Stop := "Stop Machine", "Drive 1 Brake Out" => "Drive 1 Rapid Stop", "Drive 2 Brake Out" => "Drive 2 Rapid Stop", "Drive 3 Brake Out" => "Drive 3 Rapid Stop", "Drive 4 Brake Out" => "Drive 4 Rapid Stop", "Drive 5 Brake Out" => "Drive 5 Rapid Stop", "Drive 6 Brake Out" => #"Spare Drive 6", "Drive 7 Brake Out" => #"Spare Drive 7", "Drive 8 Brake Out" => #"Spare Drive 8", "Drive 9 Brake Out" => #"Spare Drive 9", "Drive 10 Brake Out" => #"Spare Drive 10")
   END_RUNG
   // the same network as SCL:
   "EMStopDrives_Block"("Safety Callback" := "Safety Relais",
                        Direct_Stop := "Stop Machine",
                        "Drive 1 Brake Out" => "Drive 1 Rapid Stop",
                        "Drive 2 Brake Out" => "Drive 2 Rapid Stop",
                        "Drive 3 Brake Out" => "Drive 3 Rapid Stop",
                        "Drive 4 Brake Out" => "Drive 4 Rapid Stop",
                        "Drive 5 Brake Out" => "Drive 5 Rapid Stop",
                        "Drive 6 Brake Out" => #"Spare Drive 6",
                        "Drive 7 Brake Out" => #"Spare Drive 7",
                        "Drive 8 Brake Out" => #"Spare Drive 8",
                        "Drive 9 Brake Out" => #"Spare Drive 9",
                        "Drive 10 Brake Out" => #"Spare Drive 10");
END_REGION

REGION Network 11: Machine RUN
   // Function Block for System RUN, this will run the machine in automatic mode.
   // Input config is as follows:
   // - Safety Relais Contact - This input is for checking if the safety is oké, otherwise it's not possible to switch on the machine in automatic mode.
   // - Stop Machine NC Contact is the Input for the Stop button.
   // - Fill Magazine Contact is the input for the Magazine empty feedback error signal - This signal needs to be high, otherwise it's not possible to switch to automatic mode.
   // - Start Machine NO Contact is the input for Start button.
   RUNG wire#powerrail
      "SystemRUN_Block"("Safety Relais Contact" := "Safety Relais", "Stop Machine NC Contact" := "Stop Machine", "Fill Magzine Contact" := "Trechter_Bijvullen_Haltveroorzaker", "Start Machine NO Contact" := "Start Machine", "Run Output Lamp" => "LED RUN")
   END_RUNG
   // the same network as SCL:
   "SystemRUN_Block"("Safety Relais Contact" := "Safety Relais",
                     "Stop Machine NC Contact" := "Stop Machine",
                     "Fill Magzine Contact" := "Trechter_Bijvullen_Haltveroorzaker",
                     "Start Machine NO Contact" := "Start Machine",
                     "Run Output Lamp" => "LED RUN");
END_REGION

REGION Network 12: Start Infeed Belt Before Program Selection
   // This function block start the infeed belt before there's program selection. This is configured because in this way it's possible to start the machine without program selection. So products are not getting stuck on the transistion between the production line and the machine infeed belt.
   RUNG wire#powerrail
      "StartInfeedBelt_FBD"(SystemRun_Command := "Systeem RUN")
   END_RUNG
   // the same network as SCL:
   "StartInfeedBelt_FBD"(SystemRun_Command := "Systeem RUN");
END_REGION

REGION Network 13: +MC-21K11:5 - LED Programma 1
   // This network manages the selection of Program 1. It's a bit unorganized, but i'll edited it later on. Important, the move posions are not used! Axis 3 uses the movve position from the PositionManagement DB instead of these parameters!!
   RUNG wire#powerrail
      Contact( "Safety Relais" )
      I_Contact( "Noodsleutel(1)" )
      wire#w1
      I_Contact( "HMI_StartProgram" )
      Contact( "Programma 1" )
      I_Contact( "Programma 3" )
      wire#w2
      Coil( "LED Programma 1" )
      Contact( "Systeem RUN" )
      "3 - Prog. 1"(Axis_3_MovePosition1 := 0.0, Axis_3_MovePosition2 := 0.0, Axis_On_Pos_1 => "PLCMemory".ProductBuffer.RestFeedback, Axis_On_Pos_2 => "PLCMemory".ProductBuffer.MoveFeedback)
   END_RUNG
   RUNG wire#w1
      Contact( "HMI_StartProgram" )
      Contact( "HMI_StartProgram1" )
   END_RUNG wire#w2
   // the same network as SCL:
   "LED Programma 1" := "Safety Relais" AND NOT "Noodsleutel(1)" AND ((NOT "HMI_StartProgram" AND "Programma 1" AND NOT "Programma 3") OR ("HMI_StartProgram" AND "HMI_StartProgram1"));
   IF "LED Programma 1" AND "Systeem RUN" THEN
       "3 - Prog. 1"(Axis_3_MovePosition1 := 0.0,
                     Axis_3_MovePosition2 := 0.0,
                     Axis_On_Pos_1 => "PLCMemory".ProductBuffer.RestFeedback,
                     Axis_On_Pos_2 => "PLCMemory".ProductBuffer.MoveFeedback);
   END_IF;
END_REGION

REGION Network 14: +MC-21K11:2 - LED Programma 2
   // This network manages the selection of Program 2. It's a bit unorganized, but i'll edited it later on. Important, the move posions are not used! Axis 3 uses the movve position from the PositionManagement DB instead of these parameters!!
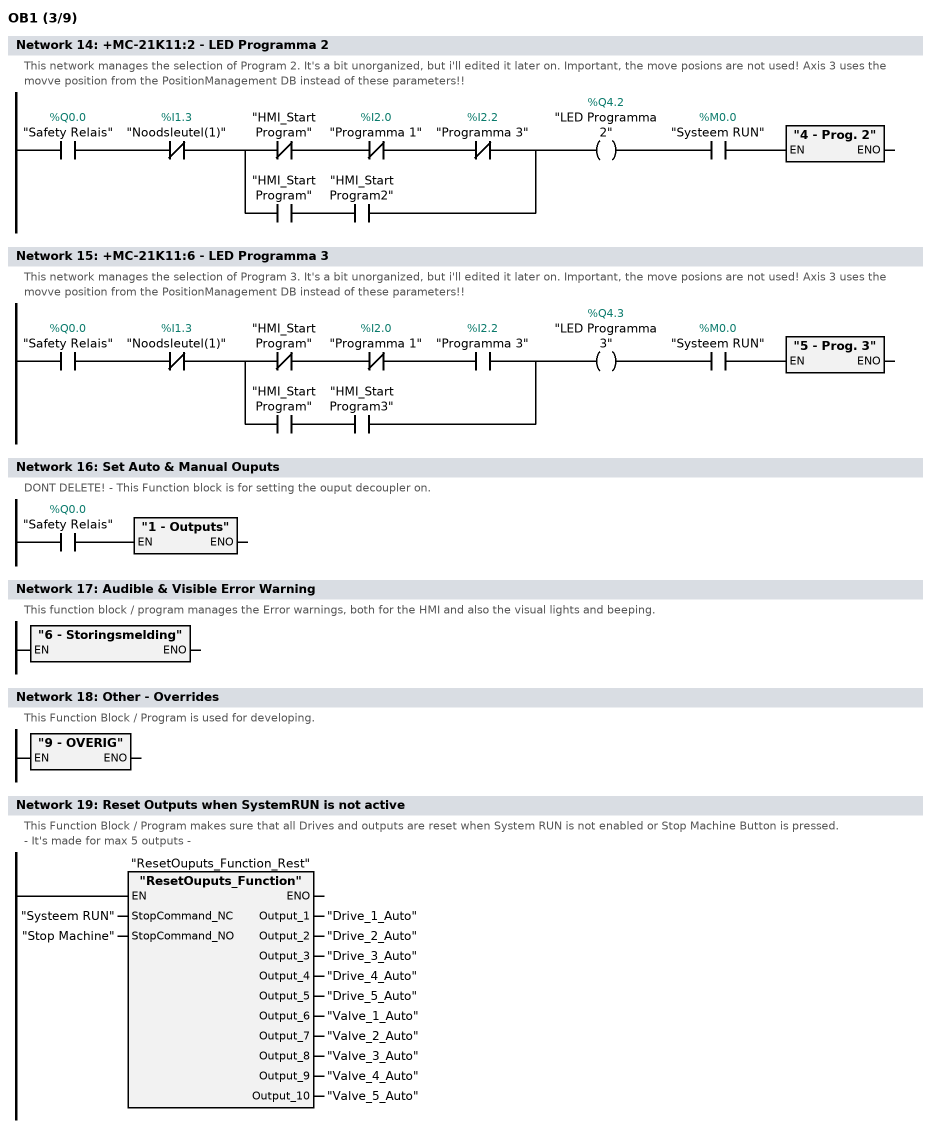
   RUNG wire#powerrail
      Contact( "Safety Relais" )
      I_Contact( "Noodsleutel(1)" )
      wire#w1
      I_Contact( "HMI_StartProgram" )
      I_Contact( "Programma 1" )
      I_Contact( "Programma 3" )
      wire#w2
      Coil( "LED Programma 2" )
      Contact( "Systeem RUN" )
      "4 - Prog. 2"()
   END_RUNG
   RUNG wire#w1
      Contact( "HMI_StartProgram" )
      Contact( "HMI_StartProgram2" )
   END_RUNG wire#w2
   // the same network as SCL:
   "LED Programma 2" := "Safety Relais" AND NOT "Noodsleutel(1)" AND ((NOT "HMI_StartProgram" AND NOT "Programma 1" AND NOT "Programma 3") OR ("HMI_StartProgram" AND "HMI_StartProgram2"));
   IF "LED Programma 2" AND "Systeem RUN" THEN "4 - Prog. 2"(); END_IF;
END_REGION

REGION Network 15: +MC-21K11:6 - LED Programma 3
   // This network manages the selection of Program 3. It's a bit unorganized, but i'll edited it later on. Important, the move posions are not used! Axis 3 uses the movve position from the PositionManagement DB instead of these parameters!!
   RUNG wire#powerrail
      Contact( "Safety Relais" )
      I_Contact( "Noodsleutel(1)" )
      wire#w1
      I_Contact( "HMI_StartProgram" )
      I_Contact( "Programma 1" )
      Contact( "Programma 3" )
      wire#w2
      Coil( "LED Programma 3" )
      Contact( "Systeem RUN" )
      "5 - Prog. 3"()
   END_RUNG
   RUNG wire#w1
      Contact( "HMI_StartProgram" )
      Contact( "HMI_StartProgram3" )
   END_RUNG wire#w2
   // the same network as SCL:
   "LED Programma 3" := "Safety Relais" AND NOT "Noodsleutel(1)" AND ((NOT "HMI_StartProgram" AND NOT "Programma 1" AND "Programma 3") OR ("HMI_StartProgram" AND "HMI_StartProgram3"));
   IF "LED Programma 3" AND "Systeem RUN" THEN "5 - Prog. 3"(); END_IF;
END_REGION

REGION Network 16: Set Auto & Manual Ouputs
   // DONT DELETE! - This Function block is for setting the ouput decoupler on.
   RUNG wire#powerrail
      Contact( "Safety Relais" )
      "1 - Outputs"()
   END_RUNG
   // the same network as SCL:
   IF "Safety Relais" THEN "1 - Outputs"(); END_IF;
END_REGION

REGION Network 17: Audible & Visible Error Warning
   // This function block / program manages the Error warnings, both for the HMI and also the visual lights and beeping.
   RUNG wire#powerrail
      "6 - Storingsmelding"()
   END_RUNG
   // the same network as SCL:
   "6 - Storingsmelding"();
END_REGION

REGION Network 18: Other - Overrides
   // This Function Block / Program is used for developing.
   RUNG wire#powerrail
      "9 - OVERIG"()
   END_RUNG
   // the same network as SCL:
   "9 - OVERIG"();
END_REGION

REGION Network 19: Reset Outputs when SystemRUN is not active
   // This Function Block / Program makes sure that all Drives and outputs are reset when System RUN is not enabled or Stop Machine Button is pressed. 
   // - It's made for max 5 outputs -
   RUNG wire#powerrail
      "ResetOuputs_Function_Rest"(StopCommand_NC := "Systeem RUN", StopCommand_NO := "Stop Machine", Output_1 => "Drive_1_Auto", Output_2 => "Drive_2_Auto", Output_3 => "Drive_3_Auto", Output_4 => "Drive_4_Auto", Output_5 => "Drive_5_Auto", Output_6 => "Valve_1_Auto", Output_7 => "Valve_2_Auto", Output_8 => "Valve_3_Auto", Output_9 => "Valve_4_Auto", Output_10 => "Valve_5_Auto")
   END_RUNG
   // the same network as SCL:
   "ResetOuputs_Function_Rest"(StopCommand_NC := "Systeem RUN",   // "ResetOuputs_Function"
                           StopCommand_NO := "Stop Machine",
                           Output_1 => "Drive_1_Auto",
                           Output_2 => "Drive_2_Auto",
                           Output_3 => "Drive_3_Auto",
                           Output_4 => "Drive_4_Auto",
                           Output_5 => "Drive_5_Auto",
                           Output_6 => "Valve_1_Auto",
                           Output_7 => "Valve_2_Auto",
                           Output_8 => "Valve_3_Auto",
                           Output_9 => "Valve_4_Auto",
                           Output_10 => "Valve_5_Auto");
END_REGION

REGION Network 20: SCL Testing block
   // This Function Block / Program is used for developing or testing.
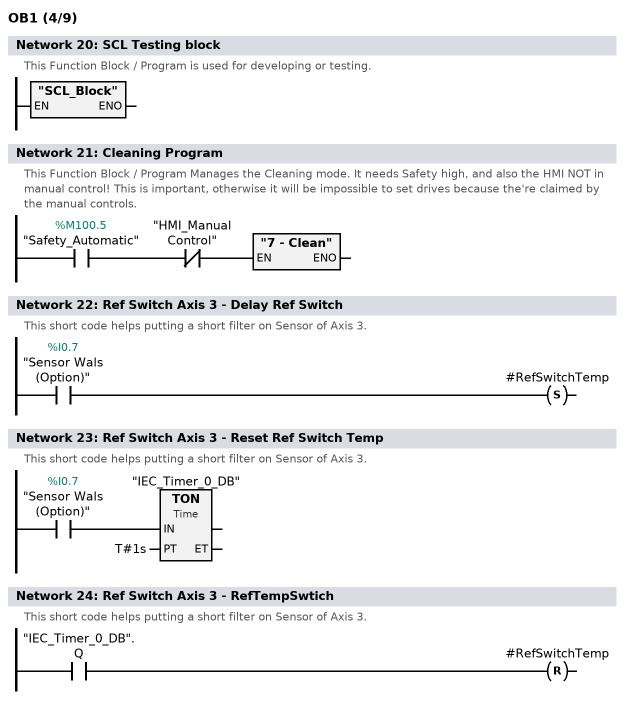
   RUNG wire#powerrail
      "SCL_Block"()
   END_RUNG
   // the same network as SCL:
   "SCL_Block"();
END_REGION

REGION Network 21: Cleaning Program
   // This Function Block / Program Manages the Cleaning mode. It needs Safety high, and also the HMI NOT in manual control! This is important, otherwise it will be impossible to set drives because the're claimed by the manual controls.
   RUNG wire#powerrail
      Contact( "Safety_Automatic" )
      I_Contact( "HMI_ManualControl" )
      "7 - Clean"()
   END_RUNG
   // the same network as SCL:
   IF "Safety_Automatic" AND NOT "HMI_ManualControl" THEN "7 - Clean"(); END_IF;
END_REGION

REGION Network 22: Ref Switch Axis 3 - Delay Ref Switch
   // This short code helps putting a short filter on Sensor of Axis 3.
   RUNG wire#powerrail
      Contact( "Sensor Wals (Option)" )
      S_Coil( #RefSwitchTemp )
   END_RUNG
   // the same network as SCL:
   IF "Sensor Wals (Option)" THEN #RefSwitchTemp := TRUE; END_IF;
END_REGION

REGION Network 23: Ref Switch Axis 3 - Reset Ref Switch Temp
   // This short code helps putting a short filter on Sensor of Axis 3.
   RUNG wire#powerrail
      Contact( "Sensor Wals (Option)" )
      { S7_Templates := "time_type := Time" } "IEC_Timer_0_DB".TON(pt := T#1s, et =>)
   END_RUNG
   // the same network as SCL:
   "IEC_Timer_0_DB".TON(IN := "Sensor Wals (Option)", PT := T#1s);
END_REGION

REGION Network 24: Ref Switch Axis 3 - RefTempSwtich
   // This short code helps putting a short filter on Sensor of Axis 3.
   RUNG wire#powerrail
      Contact( "IEC_Timer_0_DB".Q )
      R_Coil( #RefSwitchTemp )
   END_RUNG
   // the same network as SCL:
   IF "IEC_Timer_0_DB".Q THEN #RefSwitchTemp := FALSE; END_IF;
END_REGION

REGION Network 25: Drive Manager Axis 3
   // This is the Drive Manager function block, it controls the Asynchronous Servo Axis combined with an Siko IG06 Encoder. More about this can be found on the wiki page on Notion.
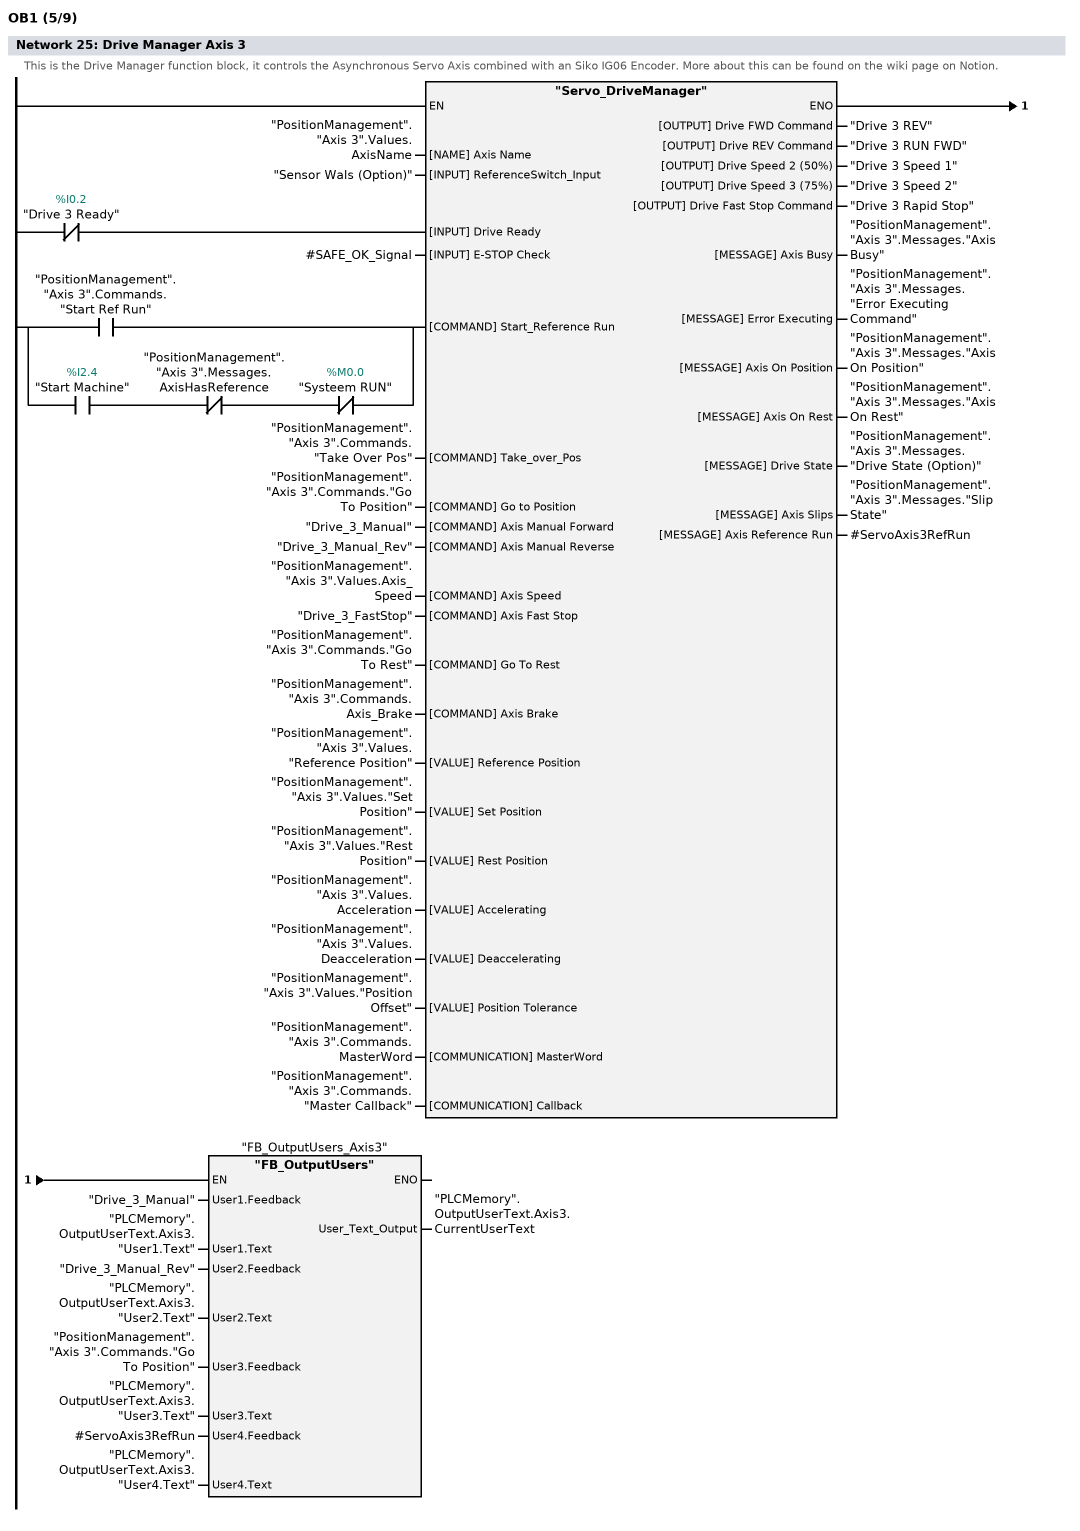
   RUNG wire#powerrail
      "Servo_DriveManager"("[INPUT] Drive Ready" := wire#w1, "[COMMAND] Start_Reference Run" := wire#w2, "[NAME] Axis Name" := "PositionManagement"."Axis 3".Values.AxisName, "[INPUT] ReferenceSwitch_Input" := "Sensor Wals (Option)", "[INPUT] E-STOP Check" := #SAFE_OK_Signal, "[COMMAND] Take_over_Pos" := "PositionManagement"."Axis 3".Commands."Take Over Pos", "[COMMAND] Go to Position" := "PositionManagement"."Axis 3".Commands."Go To Position", "[COMMAND] Axis Manual Forward" := "Drive_3_Manual", "[COMMAND] Axis Manual Reverse" := "Drive_3_Manual_Rev", "[COMMAND] Axis Speed" := "PositionManagement"."Axis 3".Values.Axis_Speed, "[COMMAND] Axis Fast Stop" := "Drive_3_FastStop", "[COMMAND] Go To Rest" := "PositionManagement"."Axis 3".Commands."Go To Rest", "[COMMAND] Axis Brake" := "PositionManagement"."Axis 3".Commands.Axis_Brake, "[VALUE] Reference Position" := "PositionManagement"."Axis 3".Values."Reference Position", "[VALUE] Set Position" := "PositionManagement"."Axis 3".Values."Set Position", "[VALUE] Rest Position" := "PositionManagement"."Axis 3".Values."Rest Position", "[VALUE] Accelerating" := "PositionManagement"."Axis 3".Values.Acceleration, "[VALUE] Deaccelerating" := "PositionManagement"."Axis 3".Values.Deacceleration, "[VALUE] Position Tolerance" := "PositionManagement"."Axis 3".Values."Position Offset", "[COMMUNICATION] MasterWord" := "PositionManagement"."Axis 3".Commands.MasterWord, "[COMMUNICATION] Callback" := "PositionManagement"."Axis 3".Commands."Master Callback", "[OUTPUT] Drive FWD Command" => "Drive 3 REV", "[OUTPUT] Drive REV Command" => "Drive 3 RUN FWD", "[OUTPUT] Drive Speed 2 (50%)" => "Drive 3 Speed 1", "[OUTPUT] Drive Speed 3 (75%)" => "Drive 3 Speed 2", "[OUTPUT] Drive Fast Stop Command" => "Drive 3 Rapid Stop", "[MESSAGE] Axis Busy" => "PositionManagement"."Axis 3".Messages."Axis Busy", "[MESSAGE] Error Executing" => "PositionManagement"."Axis 3".Messages."Error Executing Command", "[MESSAGE] Axis On Position" => "PositionManagement"."Axis 3".Messages."Axis On Position", "[MESSAGE] Axis On Rest" => "PositionManagement"."Axis 3".Messages."Axis On Rest", "[MESSAGE] Drive State" => "PositionManagement"."Axis 3".Messages."Drive State (Option)", "[MESSAGE] Axis Slips" => "PositionManagement"."Axis 3".Messages."Slip State", "[MESSAGE] Axis Reference Run" => #ServoAxis3RefRun)
      "FB_OutputUsers_Axis3"("User1.Feedback" := "Drive_3_Manual", "User1.Text" := "PLCMemory".OutputUserText.Axis3."User1.Text", "User2.Feedback" := "Drive_3_Manual_Rev", "User2.Text" := "PLCMemory".OutputUserText.Axis3."User2.Text", "User3.Feedback" := "PositionManagement"."Axis 3".Commands."Go To Position", "User3.Text" := "PLCMemory".OutputUserText.Axis3."User3.Text", "User4.Feedback" := #ServoAxis3RefRun, "User4.Text" := "PLCMemory".OutputUserText.Axis3."User4.Text", User_Text_Output => "PLCMemory".OutputUserText.Axis3.CurrentUserText)
   END_RUNG
   RUNG wire#powerrail
      I_Contact( "Drive 3 Ready" )
   END_RUNG wire#w1
   RUNG wire#powerrail
      Contact( "PositionManagement"."Axis 3".Commands."Start Ref Run" )
   END_RUNG wire#w2
   RUNG wire#powerrail
      Contact( "Start Machine" )
      I_Contact( "PositionManagement"."Axis 3".Messages.AxisHasReference )
      I_Contact( "Systeem RUN" )
   END_RUNG wire#w2
   // the same network as SCL:
   "Servo_DriveManager"("[NAME] Axis Name" := "PositionManagement"."Axis 3".Values.AxisName,
                        "[INPUT] ReferenceSwitch_Input" := "Sensor Wals (Option)",
                        "[INPUT] Drive Ready" := NOT "Drive 3 Ready",
                        "[INPUT] E-STOP Check" := #SAFE_OK_Signal,
                        "[COMMAND] Start_Reference Run" := "PositionManagement"."Axis 3".Commands."Start Ref Run" OR ("Start Machine" AND NOT "PositionManagement"."Axis 3".Messages.AxisHasReference AND NOT "Systeem RUN"),
                        "[COMMAND] Take_over_Pos" := "PositionManagement"."Axis 3".Commands."Take Over Pos",
                        "[COMMAND] Go to Position" := "PositionManagement"."Axis 3".Commands."Go To Position",
                        "[COMMAND] Axis Manual Forward" := "Drive_3_Manual",
                        "[COMMAND] Axis Manual Reverse" := "Drive_3_Manual_Rev",
                        "[COMMAND] Axis Speed" := "PositionManagement"."Axis 3".Values.Axis_Speed,
                        "[COMMAND] Axis Fast Stop" := "Drive_3_FastStop",
                        "[COMMAND] Go To Rest" := "PositionManagement"."Axis 3".Commands."Go To Rest",
                        "[COMMAND] Axis Brake" := "PositionManagement"."Axis 3".Commands.Axis_Brake,
                        "[VALUE] Reference Position" := "PositionManagement"."Axis 3".Values."Reference Position",
                        "[VALUE] Set Position" := "PositionManagement"."Axis 3".Values."Set Position",
                        "[VALUE] Rest Position" := "PositionManagement"."Axis 3".Values."Rest Position",
                        "[VALUE] Accelerating" := "PositionManagement"."Axis 3".Values.Acceleration,
                        "[VALUE] Deaccelerating" := "PositionManagement"."Axis 3".Values.Deacceleration,
                        "[VALUE] Position Tolerance" := "PositionManagement"."Axis 3".Values."Position Offset",
                        "[COMMUNICATION] MasterWord" := "PositionManagement"."Axis 3".Commands.MasterWord,
                        "[COMMUNICATION] Callback" := "PositionManagement"."Axis 3".Commands."Master Callback",
                        "[OUTPUT] Drive FWD Command" => "Drive 3 REV",
                        "[OUTPUT] Drive REV Command" => "Drive 3 RUN FWD",
                        "[OUTPUT] Drive Speed 2 (50%)" => "Drive 3 Speed 1",
                        "[OUTPUT] Drive Speed 3 (75%)" => "Drive 3 Speed 2",
                        "[OUTPUT] Drive Fast Stop Command" => "Drive 3 Rapid Stop",
                        "[MESSAGE] Axis Busy" => "PositionManagement"."Axis 3".Messages."Axis Busy",
                        "[MESSAGE] Error Executing" => "PositionManagement"."Axis 3".Messages."Error Executing Command",
                        "[MESSAGE] Axis On Position" => "PositionManagement"."Axis 3".Messages."Axis On Position",
                        "[MESSAGE] Axis On Rest" => "PositionManagement"."Axis 3".Messages."Axis On Rest",
                        "[MESSAGE] Drive State" => "PositionManagement"."Axis 3".Messages."Drive State (Option)",
                        "[MESSAGE] Axis Slips" => "PositionManagement"."Axis 3".Messages."Slip State",
                        "[MESSAGE] Axis Reference Run" => #ServoAxis3RefRun,
                        ENO => #_w1);
   IF #_w1 THEN
       "FB_OutputUsers_Axis3"("User1.Feedback" := "Drive_3_Manual",   // "FB_OutputUsers"
                              "User1.Text" := "PLCMemory".OutputUserText.Axis3."User1.Text",
                              "User2.Feedback" := "Drive_3_Manual_Rev",
                              "User2.Text" := "PLCMemory".OutputUserText.Axis3."User2.Text",
                              "User3.Feedback" := "PositionManagement"."Axis 3".Commands."Go To Position",
                              "User3.Text" := "PLCMemory".OutputUserText.Axis3."User3.Text",
                              "User4.Feedback" := #ServoAxis3RefRun,
                              "User4.Text" := "PLCMemory".OutputUserText.Axis3."User4.Text",
                              User_Text_Output => "PLCMemory".OutputUserText.Axis3.CurrentUserText);
   END_IF;
END_REGION

REGION Network 26: Noodsleutel
   // This Function Block/ Program is for the use of the Noodsleutel, when this input is HIGH, the infeed conveyorbelt is only turning.
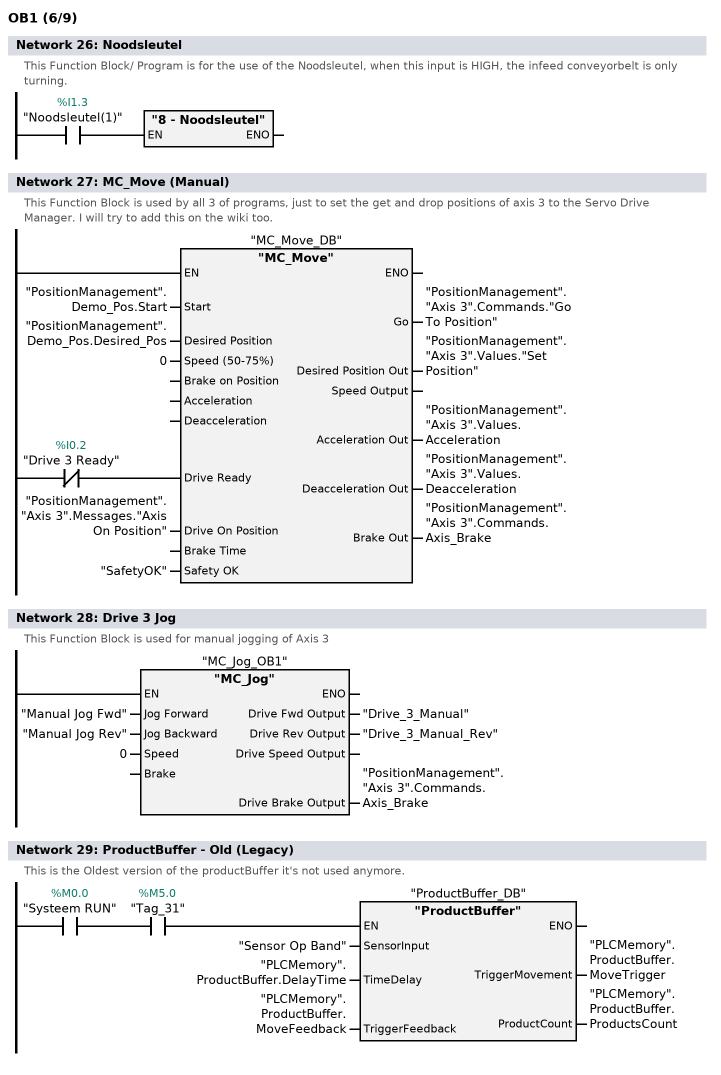
   RUNG wire#powerrail
      Contact( "Noodsleutel(1)" )
      "8 - Noodsleutel"()
   END_RUNG
   // the same network as SCL:
   IF "Noodsleutel(1)" THEN "8 - Noodsleutel"(); END_IF;
END_REGION

REGION Network 27: MC_Move (Manual)
   // This Function Block is used by all 3 of programs, just to set the get and drop positions of axis 3 to the Servo Drive Manager. I will try to add this on the wiki too.
   RUNG wire#powerrail
      "MC_Move_DB"("Drive Ready" := wire#w1, Start := "PositionManagement".Demo_Pos.Start, "Desired Position" := "PositionManagement".Demo_Pos.Desired_Pos, "Speed (50-75%)" := 0, "Brake on Position" :=, Acceleration :=, Deacceleration :=, "Drive On Position" := "PositionManagement"."Axis 3".Messages."Axis On Position", "Brake Time" :=, "Safety OK" := "SafetyOK", Go => "PositionManagement"."Axis 3".Commands."Go To Position", "Desired Position Out" => "PositionManagement"."Axis 3".Values."Set Position", "Speed Output" =>, "Acceleration Out" => "PositionManagement"."Axis 3".Values.Acceleration, "Deacceleration Out" => "PositionManagement"."Axis 3".Values.Deacceleration, "Brake Out" => "PositionManagement"."Axis 3".Commands.Axis_Brake)
   END_RUNG
   RUNG wire#powerrail
      I_Contact( "Drive 3 Ready" )
   END_RUNG wire#w1
   // the same network as SCL:
   "MC_Move_DB"(Start := "PositionManagement".Demo_Pos.Start,   // "MC_Move"
                "Desired Position" := "PositionManagement".Demo_Pos.Desired_Pos,
                "Speed (50-75%)" := 0,
                "Drive Ready" := NOT "Drive 3 Ready",
                "Drive On Position" := "PositionManagement"."Axis 3".Messages."Axis On Position",
                "Safety OK" := "SafetyOK",
                Go => "PositionManagement"."Axis 3".Commands."Go To Position",
                "Desired Position Out" => "PositionManagement"."Axis 3".Values."Set Position",
                "Acceleration Out" => "PositionManagement"."Axis 3".Values.Acceleration,
                "Deacceleration Out" => "PositionManagement"."Axis 3".Values.Deacceleration,
                "Brake Out" => "PositionManagement"."Axis 3".Commands.Axis_Brake);
END_REGION

REGION Network 28: Drive 3 Jog
   // This Function Block is used for manual jogging of Axis 3
   RUNG wire#powerrail
      "MC_Jog_OB1"("Jog Forward" := "Manual Jog Fwd", "Jog Backward" := "Manual Jog Rev", Speed := 0, Brake :=, "Drive Fwd Output" => "Drive_3_Manual", "Drive Rev Output" => "Drive_3_Manual_Rev", "Drive Speed Output" =>, "Drive Brake Output" => "PositionManagement"."Axis 3".Commands.Axis_Brake)
   END_RUNG
   // the same network as SCL:
   "MC_Jog_OB1"("Jog Forward" := "Manual Jog Fwd",   // "MC_Jog"
                "Jog Backward" := "Manual Jog Rev",
                Speed := 0,
                "Drive Fwd Output" => "Drive_3_Manual",
                "Drive Rev Output" => "Drive_3_Manual_Rev",
                "Drive Brake Output" => "PositionManagement"."Axis 3".Commands.Axis_Brake);
END_REGION

REGION Network 29: ProductBuffer - Old (Legacy)
   // This is the Oldest version of the productBuffer it's not used anymore.
   RUNG wire#powerrail
      Contact( "Systeem RUN" )
      Contact( "Tag_31" )
      "ProductBuffer_DB"(SensorInput := "Sensor Op Band", TimeDelay := "PLCMemory".ProductBuffer.DelayTime, TriggerFeedback := "PLCMemory".ProductBuffer.MoveFeedback, TriggerMovement => "PLCMemory".ProductBuffer.MoveTrigger, ProductCount => "PLCMemory".ProductBuffer.ProductsCount)
   END_RUNG
   // the same network as SCL:
   IF "Systeem RUN" AND "Tag_31" THEN
       "ProductBuffer_DB"(SensorInput := "Sensor Op Band",   // "ProductBuffer"
                          TimeDelay := "PLCMemory".ProductBuffer.DelayTime,
                          TriggerFeedback := "PLCMemory".ProductBuffer.MoveFeedback,
                          TriggerMovement => "PLCMemory".ProductBuffer.MoveTrigger,
                          ProductCount => "PLCMemory".ProductBuffer.ProductsCount);
   END_IF;
END_REGION

REGION Network 30: ProductBuffer V2 (Old - Don't use!)
   // This is Version 2 of the product buffer, and also not used anymore.
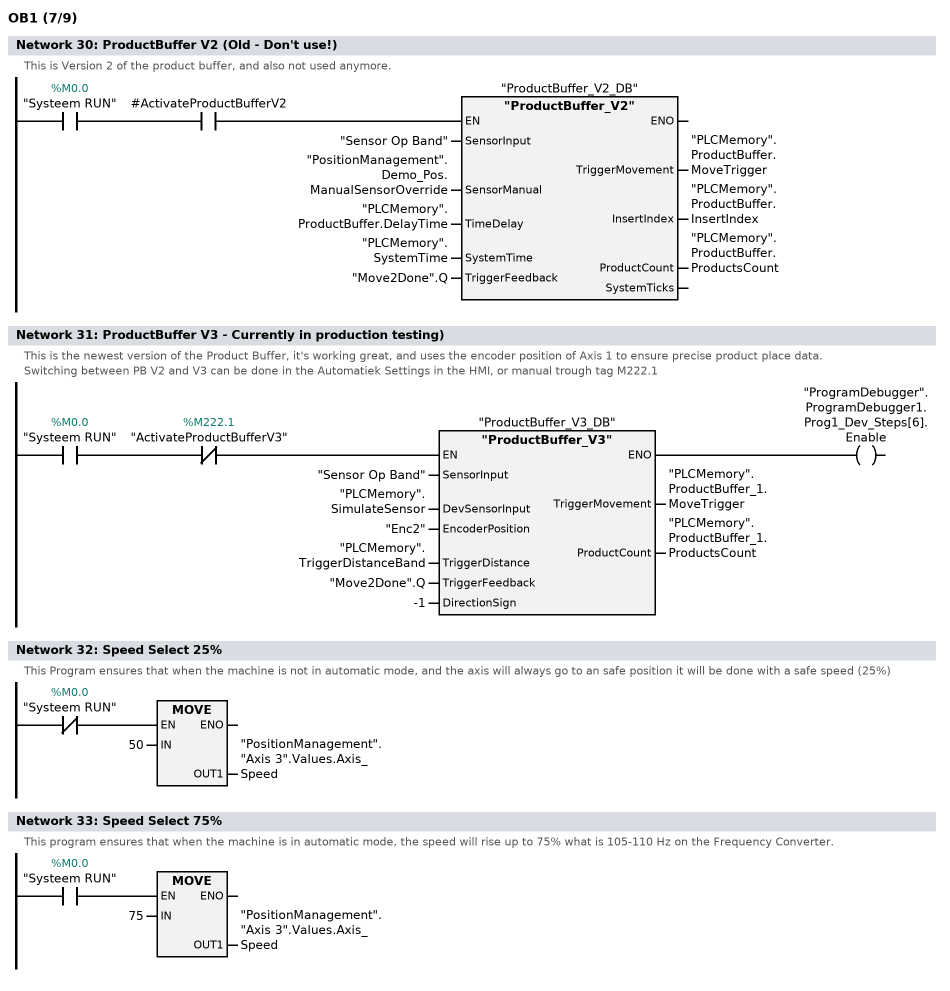
   RUNG wire#powerrail
      Contact( "Systeem RUN" )
      Contact( #ActivateProductBufferV2 )
      "ProductBuffer_V2_DB"(SensorInput := "Sensor Op Band", SensorManual := "PositionManagement".Demo_Pos.ManualSensorOverride, TimeDelay := "PLCMemory".ProductBuffer.DelayTime, SystemTime := "PLCMemory".SystemTime, TriggerFeedback := "Move2Done".Q, TriggerMovement => "PLCMemory".ProductBuffer.MoveTrigger, InsertIndex => "PLCMemory".ProductBuffer.InsertIndex, ProductCount => "PLCMemory".ProductBuffer.ProductsCount, SystemTicks =>)
   END_RUNG
   // the same network as SCL:
   IF "Systeem RUN" AND #ActivateProductBufferV2 THEN
       "ProductBuffer_V2_DB"(SensorInput := "Sensor Op Band",   // "ProductBuffer_V2"
                             SensorManual := "PositionManagement".Demo_Pos.ManualSensorOverride,
                             TimeDelay := "PLCMemory".ProductBuffer.DelayTime,
                             SystemTime := "PLCMemory".SystemTime,
                             TriggerFeedback := "Move2Done".Q,
                             TriggerMovement => "PLCMemory".ProductBuffer.MoveTrigger,
                             InsertIndex => "PLCMemory".ProductBuffer.InsertIndex,
                             ProductCount => "PLCMemory".ProductBuffer.ProductsCount);
   END_IF;
END_REGION

REGION Network 31: ProductBuffer V3 - Currently in production testing)
   // This is the newest version of the Product Buffer, it's working great, and uses the encoder position of Axis 1 to ensure precise product place data. 
   // Switching between PB V2 and V3 can be done in the Automatiek Settings in the HMI, or manual trough tag M222.1
   RUNG wire#powerrail
      Contact( "Systeem RUN" )
      I_Contact( "ActivateProductBufferV3" )
      "ProductBuffer_V3_DB"(SensorInput := "Sensor Op Band", DevSensorInput := "PLCMemory".SimulateSensor, EncoderPosition := "Enc2", TriggerDistance := "PLCMemory".TriggerDistanceBand, TriggerFeedback := "Move2Done".Q, DirectionSign := -1, TriggerMovement => "PLCMemory".ProductBuffer_1.MoveTrigger, ProductCount => "PLCMemory".ProductBuffer_1.ProductsCount)
      Coil( "ProgramDebugger".ProgramDebugger1.Prog1_Dev_Steps[6].Enable )
   END_RUNG
   // the same network as SCL:
   "ProductBuffer_V3_DB"(EN := "Systeem RUN" AND NOT "ActivateProductBufferV3",   // "ProductBuffer_V3"
                         SensorInput := "Sensor Op Band",
                         DevSensorInput := "PLCMemory".SimulateSensor,
                         EncoderPosition := "Enc2",
                         TriggerDistance := "PLCMemory".TriggerDistanceBand,
                         TriggerFeedback := "Move2Done".Q,
                         DirectionSign := -1,
                         TriggerMovement => "PLCMemory".ProductBuffer_1.MoveTrigger,
                         ProductCount => "PLCMemory".ProductBuffer_1.ProductsCount,
                         ENO => #_w1);
   "ProgramDebugger".ProgramDebugger1.Prog1_Dev_Steps[6].Enable := #_w1;
END_REGION

REGION Network 32: Speed Select 25%
   // This Program ensures that when the machine is not in automatic mode, and the axis will always go to an safe position it will be done with a safe speed (25%)
   RUNG wire#powerrail
      I_Contact( "Systeem RUN" )
      { S7_GenerateENO := "TRUE" } Move(in := 50, out1 => "PositionManagement"."Axis 3".Values.Axis_Speed)
   END_RUNG
   // the same network as SCL:
   IF NOT "Systeem RUN" THEN "PositionManagement"."Axis 3".Values.Axis_Speed := 50; END_IF;
END_REGION

REGION Network 33: Speed Select 75%
   // This program ensures that when the machine is in automatic mode, the speed will rise up to 75% what is 105-110 Hz on the Frequency Converter.
   RUNG wire#powerrail
      Contact( "Systeem RUN" )
      { S7_GenerateENO := "TRUE" } Move(in := 75, out1 => "PositionManagement"."Axis 3".Values.Axis_Speed)
   END_RUNG
   // the same network as SCL:
   IF "Systeem RUN" THEN "PositionManagement"."Axis 3".Values.Axis_Speed := 75; END_IF;
END_REGION

REGION Network 34: Encoder Band Function Block
   // This Function Block is for controlling and reading encoder data from the Axis 1 SIKO IG09 encoder. More can be found on the wiki.
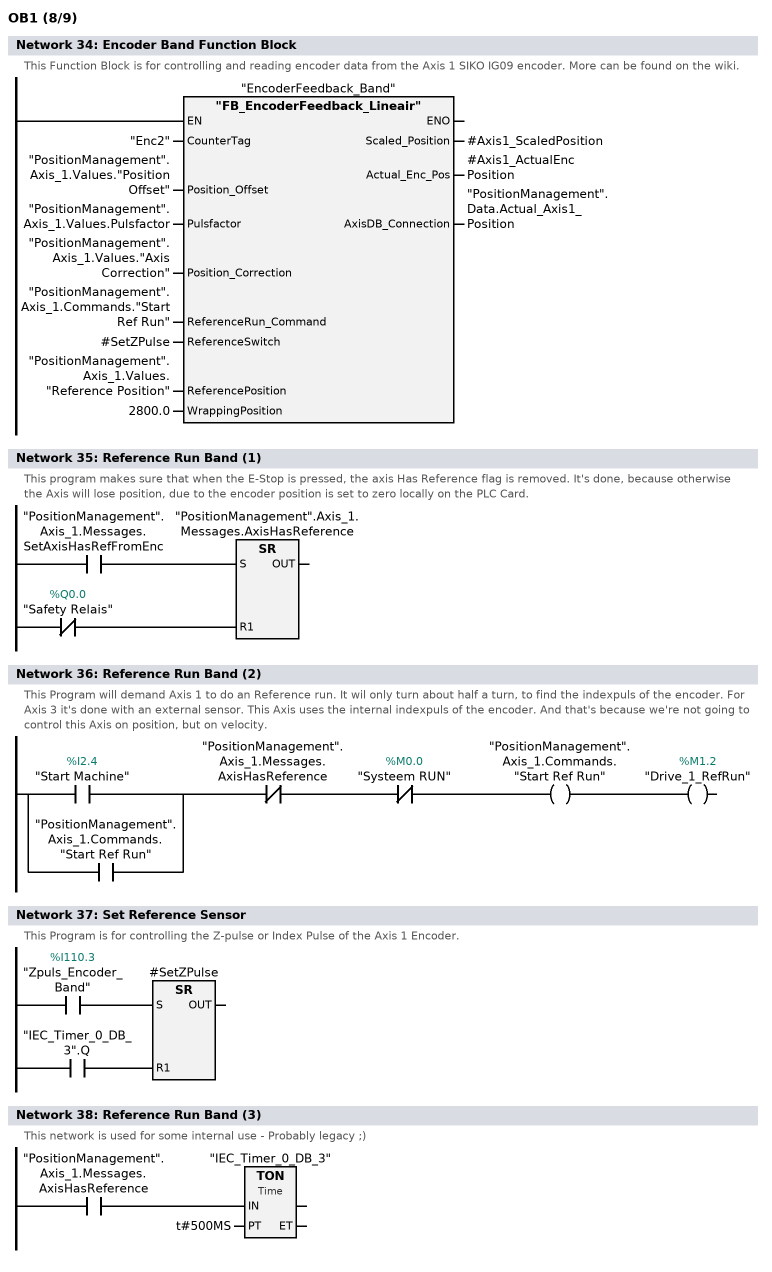
   RUNG wire#powerrail
      "EncoderFeedback_Band"(CounterTag := "Enc2", Position_Offset := "PositionManagement".Axis_1.Values."Position Offset", Pulsfactor := "PositionManagement".Axis_1.Values.Pulsfactor, Position_Correction := "PositionManagement".Axis_1.Values."Axis Correction", ReferenceRun_Command := "PositionManagement".Axis_1.Commands."Start Ref Run", ReferenceSwitch := #SetZPulse, ReferencePosition := "PositionManagement".Axis_1.Values."Reference Position", WrappingPosition := 2800.0, Scaled_Position => #Axis1_ScaledPosition, Actual_Enc_Pos => #Axis1_ActualEncPosition, AxisDB_Connection => "PositionManagement".Data.Actual_Axis1_Position)
   END_RUNG
   // the same network as SCL:
   "EncoderFeedback_Band"(CounterTag := "Enc2",   // "FB_EncoderFeedback_Lineair"
                          Position_Offset := "PositionManagement".Axis_1.Values."Position Offset",
                          Pulsfactor := "PositionManagement".Axis_1.Values.Pulsfactor,
                          Position_Correction := "PositionManagement".Axis_1.Values."Axis Correction",
                          ReferenceRun_Command := "PositionManagement".Axis_1.Commands."Start Ref Run",
                          ReferenceSwitch := #SetZPulse,
                          ReferencePosition := "PositionManagement".Axis_1.Values."Reference Position",
                          WrappingPosition := 2800.0,
                          Scaled_Position => #Axis1_ScaledPosition,
                          Actual_Enc_Pos => #Axis1_ActualEncPosition,
                          AxisDB_Connection => "PositionManagement".Data.Actual_Axis1_Position);
END_REGION

REGION Network 35: Reference Run Band (1)
   // This program makes sure that when the E-Stop is pressed, the axis Has Reference flag is removed. It's done, because otherwise the Axis will lose position, due to the encoder position is set to zero locally on the PLC Card.
   RUNG wire#powerrail
      Contact( "PositionManagement".Axis_1.Messages.SetAxisHasRefFromEnc )
      S_SR(operand := "PositionManagement".Axis_1.Messages.AxisHasReference, r1 := wire#w1)
   END_RUNG
   RUNG wire#powerrail
      I_Contact( "Safety Relais" )
   END_RUNG wire#w1
   // the same network as SCL:
   IF "PositionManagement".Axis_1.Messages.SetAxisHasRefFromEnc THEN
       "PositionManagement".Axis_1.Messages.AxisHasReference := TRUE;   // SR flip-flop
   END_IF;
   IF NOT "Safety Relais" THEN "PositionManagement".Axis_1.Messages.AxisHasReference := FALSE; END_IF;
END_REGION

REGION Network 36: Reference Run Band (2)
   // This Program will demand Axis 1 to do an Reference run. It wil only turn about half a turn, to find the indexpuls of the encoder. For Axis 3 it's done with an external sensor. This Axis uses the internal indexpuls of the encoder. And that's because we're not going to control this Axis on position, but on velocity.
   RUNG wire#powerrail
      Contact( "Start Machine" )
      wire#w1
      I_Contact( "PositionManagement".Axis_1.Messages.AxisHasReference )
      I_Contact( "Systeem RUN" )
      Coil( "PositionManagement".Axis_1.Commands."Start Ref Run" )
      Coil( "Drive_1_RefRun" )
   END_RUNG
   RUNG wire#powerrail
      Contact( "PositionManagement".Axis_1.Commands."Start Ref Run" )
   END_RUNG wire#w1
   // the same network as SCL:
   "PositionManagement".Axis_1.Commands."Start Ref Run" := ("Start Machine" OR "PositionManagement".Axis_1.Commands."Start Ref Run") AND NOT "PositionManagement".Axis_1.Messages.AxisHasReference AND NOT "Systeem RUN";
   "Drive_1_RefRun" := "PositionManagement".Axis_1.Commands."Start Ref Run";
END_REGION

REGION Network 37: Set Reference Sensor
   // This Program is for controlling the Z-pulse or Index Pulse of the Axis 1 Encoder.
   RUNG wire#powerrail
      Contact( "Zpuls_Encoder_Band" )
      S_SR(operand := #SetZPulse, r1 := wire#w1)
   END_RUNG
   RUNG wire#powerrail
      Contact( "IEC_Timer_0_DB_3".Q )
   END_RUNG wire#w1
   // the same network as SCL:
   IF "Zpuls_Encoder_Band" THEN
       #SetZPulse := TRUE;   // SR flip-flop
   END_IF;
   IF "IEC_Timer_0_DB_3".Q THEN #SetZPulse := FALSE; END_IF;
END_REGION

REGION Network 38: Reference Run Band (3)
   // This network is used for some internal use - Probably legacy ;)
   RUNG wire#powerrail
      Contact( "PositionManagement".Axis_1.Messages.AxisHasReference )
      { S7_Templates := "time_type := Time" } "IEC_Timer_0_DB_3".TON(pt := t#500MS, et =>)
   END_RUNG
   // the same network as SCL:
   "IEC_Timer_0_DB_3".TON(IN := "PositionManagement".Axis_1.Messages.AxisHasReference, PT := t#500MS);
END_REGION

REGION Network 39: SystemTime
   // This network will read the PLC Uptime. It was used for timestamp purposes.
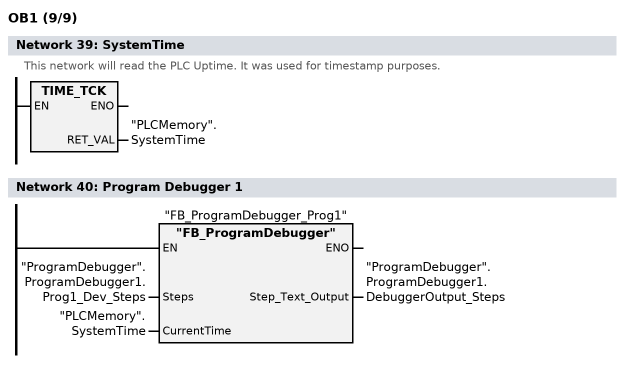
   RUNG wire#powerrail
      TIME_TCK(RET_VAL => "PLCMemory".SystemTime)
   END_RUNG
   // the same network as SCL:
   "PLCMemory".SystemTime := TIME_TCK();
END_REGION

REGION Network 40: Program Debugger 1
   RUNG wire#powerrail
      "FB_ProgramDebugger_Prog1"(Steps := "ProgramDebugger".ProgramDebugger1.Prog1_Dev_Steps, CurrentTime := "PLCMemory".SystemTime, Step_Text_Output => "ProgramDebugger".ProgramDebugger1.DebuggerOutput_Steps)
   END_RUNG
   // the same network as SCL:
   "FB_ProgramDebugger_Prog1"(Steps := "ProgramDebugger".ProgramDebugger1.Prog1_Dev_Steps,   // "FB_ProgramDebugger"
                           CurrentTime := "PLCMemory".SystemTime,
                           Step_Text_Output => "ProgramDebugger".ProgramDebugger1.DebuggerOutput_Steps);
END_REGION
END_ORGANIZATION_BLOCK

FUNCTION "SafetyFunction_Block" : Void   // FC12, LAD
VERSION : 0.1
// stored: AutoNumber true, IsIECCheckEnabled false, UDAEnableTagReadback false
   VAR_INPUT
      "ESB NC Contact" : Bool;
      "ESB NO Contact" : Bool;
      "Reset NO Contact" : Bool;
      "SAFE door 1 NC Contact" : Bool;
      "SAFE door 2 NC Contact" : Bool;
      "Safety Relais NO Contact" : Bool;
   END_VAR
   VAR_OUTPUT
      SAFE_OK_Signal : Bool;
   END_VAR
BEGIN

REGION Network 1: +MC-21K6:1 - Noodstop Circuit
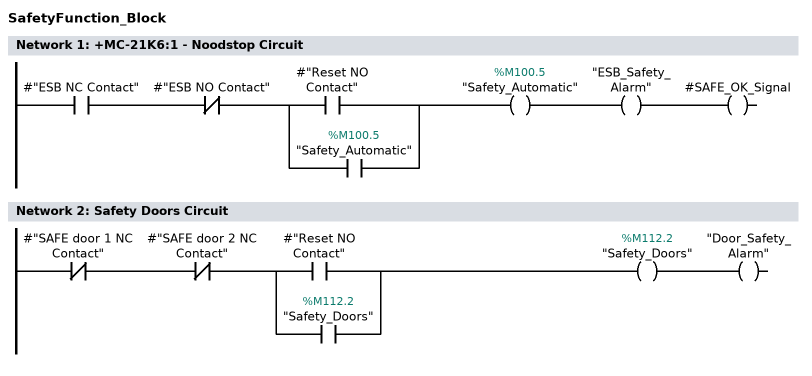
   RUNG wire#powerrail
      Contact( #"ESB NC Contact" )
      I_Contact( #"ESB NO Contact" )
      wire#w1
      Contact( #"Reset NO Contact" )
      wire#w2
      Coil( "Safety_Automatic" )
      Coil( "ESB_Safety_Alarm" )
      Coil( #SAFE_OK_Signal )
   END_RUNG
   RUNG wire#w1
      Contact( "Safety_Automatic" )
   END_RUNG wire#w2
   // the same network as SCL:
   "Safety_Automatic" := #"ESB NC Contact" AND NOT #"ESB NO Contact" AND (#"Reset NO Contact" OR "Safety_Automatic");
   "ESB_Safety_Alarm" := "Safety_Automatic";
   #SAFE_OK_Signal := "Safety_Automatic";
END_REGION

REGION Network 2: Safety Doors Circuit
   RUNG wire#powerrail
      I_Contact( #"SAFE door 1 NC Contact" )
      I_Contact( #"SAFE door 2 NC Contact" )
      wire#w1
      Contact( #"Reset NO Contact" )
      wire#w2
      Coil( "Safety_Doors" )
      Coil( "Door_Safety_Alarm" )
   END_RUNG
   RUNG wire#w1
      Contact( "Safety_Doors" )
   END_RUNG wire#w2
   // the same network as SCL:
   "Safety_Doors" := NOT #"SAFE door 1 NC Contact" AND NOT #"SAFE door 2 NC Contact" AND (#"Reset NO Contact" OR "Safety_Doors");
   "Door_Safety_Alarm" := "Safety_Doors";
END_REGION
END_FUNCTION

FUNCTION "EMStopDrives_Block" : Void   // FC14, LAD
VERSION : 0.1
// stored: AutoNumber true, IsIECCheckEnabled false, UDAEnableTagReadback false
   VAR_INPUT
      "Safety Callback" : Bool;
      Direct_Stop : Bool;
   END_VAR
   VAR_OUTPUT
      "Drive 1 Brake Out" : Bool;
      "Drive 2 Brake Out" : Bool;
      "Drive 3 Brake Out" : Bool;
      "Drive 4 Brake Out" : Bool;
      "Drive 5 Brake Out" : Bool;
      "Drive 6 Brake Out" : Bool;
      "Drive 7 Brake Out" : Bool;
      "Drive 8 Brake Out" : Bool;
      "Drive 9 Brake Out" : Bool;
      "Drive 10 Brake Out" : Bool;
   END_VAR
BEGIN

REGION Network 1: Drives Emergency Stop
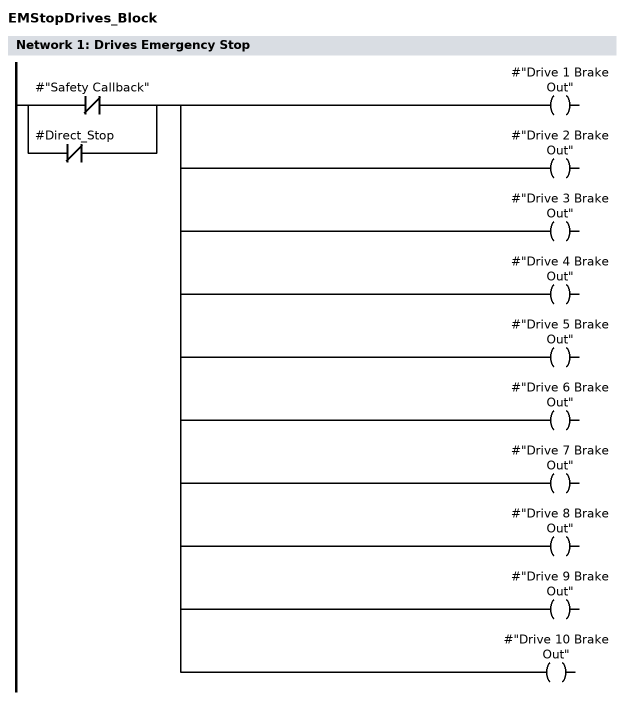
   RUNG wire#powerrail
      I_Contact( #"Safety Callback" )
      wire#w1
      Coil( #"Drive 1 Brake Out" )
   END_RUNG
   RUNG wire#powerrail
      I_Contact( #Direct_Stop )
   END_RUNG wire#w1
   RUNG wire#w1
      Coil( #"Drive 2 Brake Out" )
   END_RUNG
   RUNG wire#w1
      Coil( #"Drive 3 Brake Out" )
   END_RUNG
   RUNG wire#w1
      Coil( #"Drive 4 Brake Out" )
   END_RUNG
   RUNG wire#w1
      Coil( #"Drive 5 Brake Out" )
   END_RUNG
   RUNG wire#w1
      Coil( #"Drive 6 Brake Out" )
   END_RUNG
   RUNG wire#w1
      Coil( #"Drive 7 Brake Out" )
   END_RUNG
   RUNG wire#w1
      Coil( #"Drive 8 Brake Out" )
   END_RUNG
   RUNG wire#w1
      Coil( #"Drive 9 Brake Out" )
   END_RUNG
   RUNG wire#w1
      Coil( #"Drive 10 Brake Out" )
   END_RUNG
   // the same network as SCL:
   #"Drive 1 Brake Out" := NOT #"Safety Callback" OR NOT #Direct_Stop;
   #"Drive 2 Brake Out" := #"Drive 1 Brake Out";
   #"Drive 3 Brake Out" := #"Drive 1 Brake Out";
   #"Drive 4 Brake Out" := #"Drive 1 Brake Out";
   #"Drive 5 Brake Out" := #"Drive 1 Brake Out";
   #"Drive 6 Brake Out" := #"Drive 1 Brake Out";
   #"Drive 7 Brake Out" := #"Drive 1 Brake Out";
   #"Drive 8 Brake Out" := #"Drive 1 Brake Out";
   #"Drive 9 Brake Out" := #"Drive 1 Brake Out";
   #"Drive 10 Brake Out" := #"Drive 1 Brake Out";
END_REGION
END_FUNCTION

FUNCTION "SystemRUN_Block" : Void   // FC13, LAD
VERSION : 0.1
// stored: AutoNumber true, IsIECCheckEnabled false, UDAEnableTagReadback false
   VAR_INPUT
      "Safety Relais Contact" : Bool;
      "Stop Machine NC Contact" : Bool;
      "Fill Magzine Contact" : Bool;
      "Start Machine NO Contact" : Bool;
   END_VAR
   VAR_OUTPUT
      "Run Output Lamp" : Bool;
   END_VAR
BEGIN

REGION Network 1: Systeem RUN
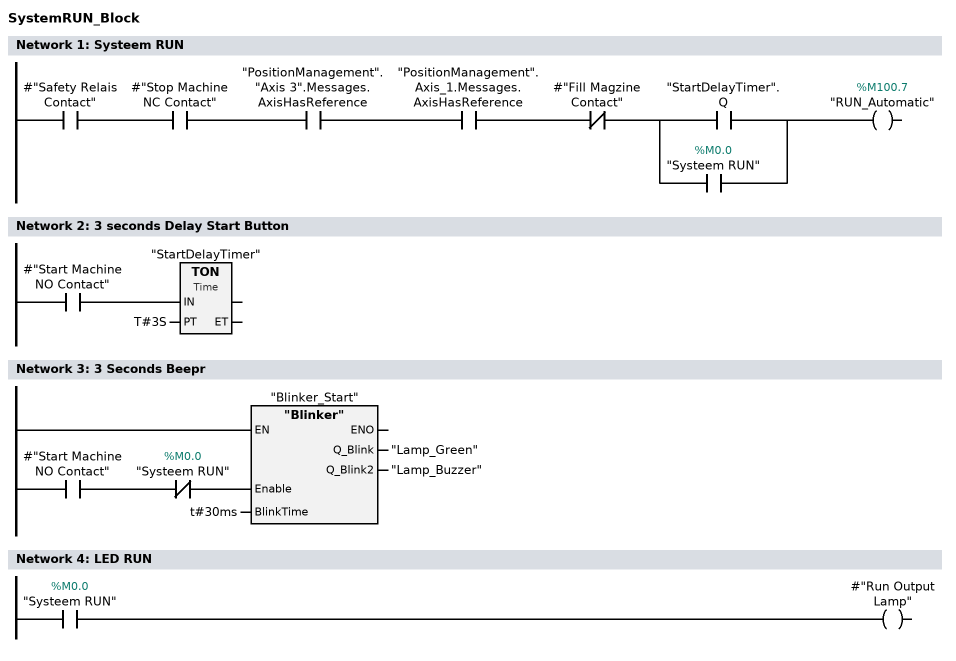
   RUNG wire#powerrail
      Contact( #"Safety Relais Contact" )
      Contact( #"Stop Machine NC Contact" )
      Contact( "PositionManagement"."Axis 3".Messages.AxisHasReference )
      Contact( "PositionManagement".Axis_1.Messages.AxisHasReference )
      I_Contact( #"Fill Magzine Contact" )
      wire#w1
      Contact( "StartDelayTimer".Q )
      wire#w2
      Coil( "RUN_Automatic" )
   END_RUNG
   RUNG wire#w1
      Contact( "Systeem RUN" )
   END_RUNG wire#w2
   // the same network as SCL:
   "RUN_Automatic" := #"Safety Relais Contact" AND #"Stop Machine NC Contact" AND "PositionManagement"."Axis 3".Messages.AxisHasReference AND "PositionManagement".Axis_1.Messages.AxisHasReference AND NOT #"Fill Magzine Contact" AND ("StartDelayTimer".Q OR "Systeem RUN");
END_REGION

REGION Network 2: 3 seconds Delay Start Button
   RUNG wire#powerrail
      Contact( #"Start Machine NO Contact" )
      { S7_Templates := "time_type := Time" } "StartDelayTimer".TON(pt := T#3S, et =>)
   END_RUNG
   // the same network as SCL:
   "StartDelayTimer".TON(IN := #"Start Machine NO Contact", PT := T#3S);
END_REGION

REGION Network 3: 3 Seconds Beepr
   RUNG wire#powerrail
      "Blinker_Start"(Enable := wire#w1, BlinkTime := t#30ms, Q_Blink => "Lamp_Green", Q_Blink2 => "Lamp_Buzzer")
   END_RUNG
   RUNG wire#powerrail
      Contact( #"Start Machine NO Contact" )
      I_Contact( "Systeem RUN" )
   END_RUNG wire#w1
   // the same network as SCL:
   "Blinker_Start"(Enable := #"Start Machine NO Contact" AND NOT "Systeem RUN",   // "Blinker"
                   BlinkTime := t#30ms,
                   Q_Blink => "Lamp_Green",
                   Q_Blink2 => "Lamp_Buzzer");
END_REGION

REGION Network 4: LED RUN
   RUNG wire#powerrail
      Contact( "Systeem RUN" )
      Coil( #"Run Output Lamp" )
   END_RUNG
   // the same network as SCL:
   #"Run Output Lamp" := "Systeem RUN";
END_REGION
END_FUNCTION

FUNCTION_BLOCK "Blinker"
{ S7_Optimized_Access := 'FALSE' }
VERSION : 0.1
   VAR_INPUT 
      Enable : Bool;
      BlinkTime : Time := T#500ms;
   END_VAR

   VAR_OUTPUT 
      Q_Blink : Bool;
      Q_Blink2 : Bool;
   END_VAR

   VAR 
      BlinkTimer {InstructionName := 'TON'; LibVersion := '1.0'; S7_SetPoint := 'False'} : TON;
   END_VAR

   VAR_TEMP 
      LastToggleTime : Time;
   END_VAR


BEGIN
	// Logica
	IF #Enable THEN
	    #BlinkTimer(IN := TRUE,
	                PT := #BlinkTime);   // Correct gebruik van PT
	    
	    IF #BlinkTimer.Q THEN
	        #Q_Blink := NOT #Q_Blink;                // Toggle uitgang
	        #Q_Blink2 := NOT #Q_Blink2;
	        #BlinkTimer(IN := FALSE,
	                    PT := #BlinkTime); // Reset timer (verplicht opnieuw PT meegeven)
	    END_IF;
	    
	ELSE
	    #BlinkTimer(IN := FALSE,
	                PT := #BlinkTime);  // Timer uitzetten
	    #Q_Blink := FALSE; // Uitgang terug laag
	    #Q_Blink2 := FALSE;
	END_IF;
END_FUNCTION_BLOCK

FUNCTION "StartInfeedBelt_FBD" : Void   // FC11, FBD
TITLE = StartInfeedBelt
VERSION : 0.1
// stored: AutoNumber true, IsIECCheckEnabled false, UDAEnableTagReadback false
   VAR_INPUT
      SystemRun_Command : Bool;
   END_VAR
BEGIN

REGION Network 2: Aanvoerband (1) - Aansturen
   // This block sets an starttimer on Drive 1
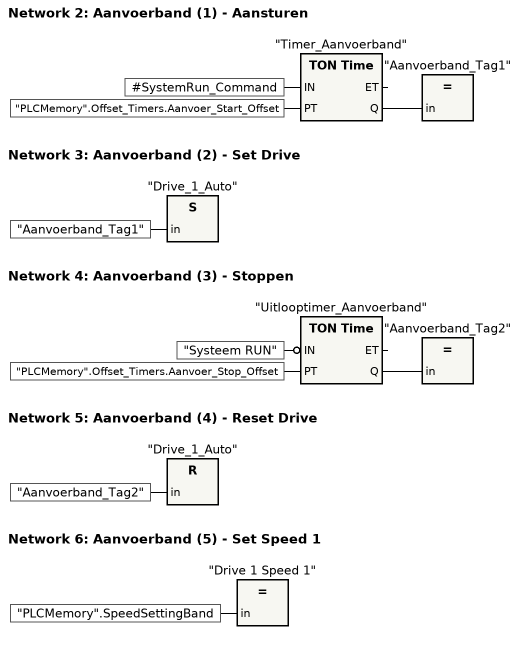
   "Timer_Aanvoerband".TON(IN := #SystemRun_Command, PT := "PLCMemory".Offset_Timers.Aanvoer_Start_Offset);
   "Aanvoerband_Tag1" := "Timer_Aanvoerband".Q;
END_REGION

REGION Network 3: Aanvoerband (2) - Set Drive
   // This block sets Drive 1 Auto signal
   IF "Aanvoerband_Tag1" THEN "Drive_1_Auto" := TRUE; END_IF;
END_REGION

REGION Network 4: Aanvoerband (3) - Stoppen
   // This block sets an End timer on Drive 1
   "Uitlooptimer_Aanvoerband".TON(IN := NOT "Systeem RUN", PT := "PLCMemory".Offset_Timers.Aanvoer_Stop_Offset);
   "Aanvoerband_Tag2" := "Uitlooptimer_Aanvoerband".Q;
END_REGION

REGION Network 5: Aanvoerband (4) - Reset Drive
   // This block resets Drive 1 Auto
   IF "Aanvoerband_Tag2" THEN "Drive_1_Auto" := FALSE; END_IF;
END_REGION

REGION Network 6: Aanvoerband (5) - Set Speed 1
   // This block sets the speed for Drive 1
   "Drive 1 Speed 1" := "PLCMemory".SpeedSettingBand;
END_REGION
END_FUNCTION

FUNCTION "3 - Prog. 1" : Void   // FC1, LAD
TITLE = System Program 1
VERSION : 0.1
// DF
// stored: AutoNumber true, IsIECCheckEnabled false, UDAEnableTagReadback false
   VAR_INPUT
      Axis_3_MovePosition1 : Real;
      Axis_3_MovePosition2 : Real;
   END_VAR
   VAR_OUTPUT
      Axis_On_Pos_1 : Bool;
      Axis_On_Pos_2 : Bool;
   END_VAR
   VAR_TEMP
      TempProdCounter : Int;
      Temp_ProductsToProduce : Bool;
      TimerRunning : Bool;
      ProduceContact : Bool;
      Move2Done : Bool;
      SRWals : Bool;
      Move2Busy : Bool;
      SR_Move2 : Bool;
      Move1Busy : Bool;
      P_TRIG_SnrBand : Bool;
      Temp1 : Bool;
      Min_Pos_1 : Real;
      Max_Pos_1 : Real;
      Min_Pos_2 : Real;
      Max_Pos_2 : Real;
      SR_Move3 : Bool;
      SR_Move1 : Bool;
      AxisToRest : Bool;
      SubDone : Bool;
      P_Trig_ProBehWals : Bool;
      ProductsBehindWals : Int;
      ProductBehindWals : Bool;
      AandrukCilindersOut : Bool;
      Retourband_Delayed : Bool;
      BlowOff_Activated : Bool;
      Pos2_Done : Bool;
      Pos1_Done : Bool;
      ToWaitPosition : Bool;
      BlowOffConf : Bool;
      PTrig_Blow : Bool;
      Move2Done_2 : Bool;
      GoToMove2Pos : Bool;
      GoToMove2 : Bool;
      Democoil_Nofunction : Bool;
      StartBlowOff : Bool;
      BlowOffTimer : Bool;
      Democoil : Bool;
      WaitForMove2 : Bool;
      SRBlowOff : Bool;
      PTRigBlowOf : Bool;
      SRTriggerBlowing : Bool;
      Debugger1RS : Bool;
   END_VAR
   VAR_TEMP   // added for the SCL form of the ladder/FBD networks
      _w1 : Bool;
   END_VAR
BEGIN

REGION Network 1: Debugger Trilgoten (1)
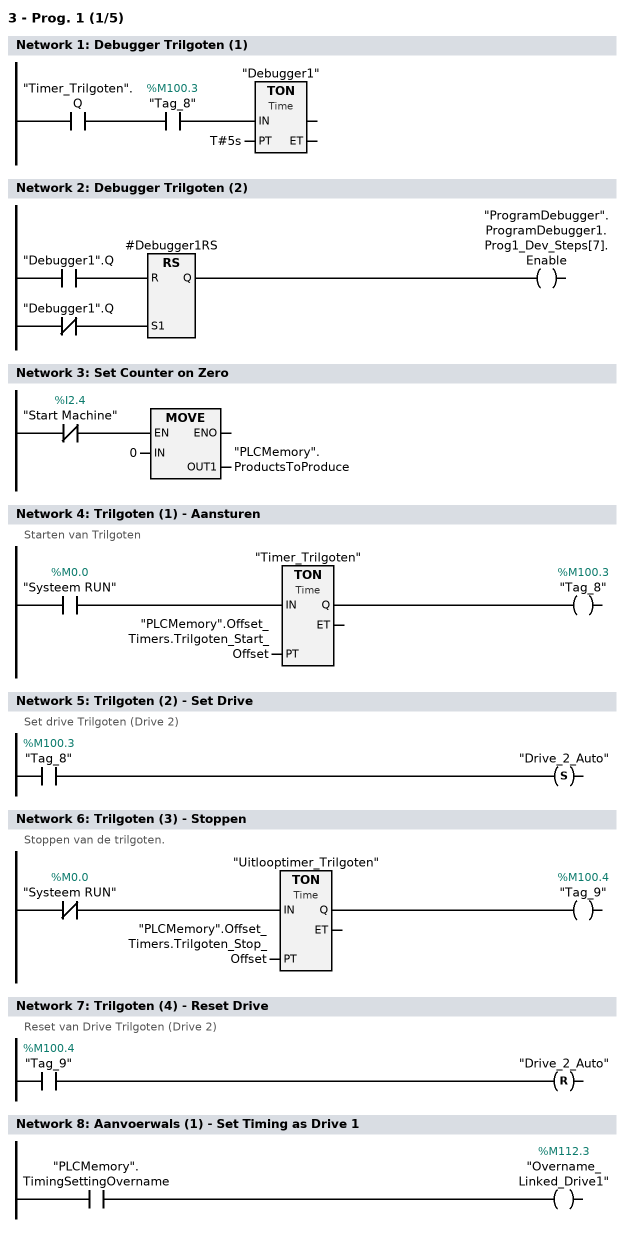
   RUNG wire#powerrail
      Contact( "Timer_Trilgoten".Q )
      Contact( "Tag_8" )
      { S7_Templates := "time_type := Time" } "Debugger1".TON(pt := T#5s, et =>)
   END_RUNG
   // the same network as SCL:
   "Debugger1".TON(IN := "Timer_Trilgoten".Q AND "Tag_8", PT := T#5s);
END_REGION

REGION Network 2: Debugger Trilgoten (2)
   RUNG wire#powerrail
      Contact( "Debugger1".Q )
      S_RS(operand := #Debugger1RS, s1 := wire#w1)
      Coil( "ProgramDebugger".ProgramDebugger1.Prog1_Dev_Steps[7].Enable )
   END_RUNG
   RUNG wire#powerrail
      I_Contact( "Debugger1".Q )
   END_RUNG wire#w1
   // the same network as SCL:
   IF "Debugger1".Q THEN
       #Debugger1RS := FALSE;   // RS flip-flop
   END_IF;
   IF NOT "Debugger1".Q THEN #Debugger1RS := TRUE; END_IF;
   "ProgramDebugger".ProgramDebugger1.Prog1_Dev_Steps[7].Enable := #Debugger1RS;
END_REGION

REGION Network 3: Set Counter on Zero
   RUNG wire#powerrail
      I_Contact( "Start Machine" )
      { S7_GenerateENO := "TRUE" } Move(in := 0, out1 => "PLCMemory".ProductsToProduce)
   END_RUNG
   // the same network as SCL:
   IF NOT "Start Machine" THEN "PLCMemory".ProductsToProduce := 0; END_IF;
END_REGION

REGION Network 4: Trilgoten (1) - Aansturen
   // Starten van Trilgoten
   RUNG wire#powerrail
      Contact( "Systeem RUN" )
      { S7_Templates := "time_type := Time" } "Timer_Trilgoten".TON(pt := "PLCMemory".Offset_Timers.Trilgoten_Start_Offset, et =>)
      Coil( "Tag_8" )
   END_RUNG
   // the same network as SCL:
   "Timer_Trilgoten".TON(IN := "Systeem RUN", PT := "PLCMemory".Offset_Timers.Trilgoten_Start_Offset);
   "Tag_8" := "Timer_Trilgoten".Q;
END_REGION

REGION Network 5: Trilgoten (2) - Set Drive
   // Set drive Trilgoten (Drive 2)
   RUNG wire#powerrail
      Contact( "Tag_8" )
      S_Coil( "Drive_2_Auto" )
   END_RUNG
   // the same network as SCL:
   IF "Tag_8" THEN "Drive_2_Auto" := TRUE; END_IF;
END_REGION

REGION Network 6: Trilgoten (3) - Stoppen
   // Stoppen van de trilgoten.
   RUNG wire#powerrail
      I_Contact( "Systeem RUN" )
      { S7_Templates := "time_type := Time" } "Uitlooptimer_Trilgoten".TON(pt := "PLCMemory".Offset_Timers.Trilgoten_Stop_Offset, et =>)
      Coil( "Tag_9" )
   END_RUNG
   // the same network as SCL:
   "Uitlooptimer_Trilgoten".TON(IN := NOT "Systeem RUN", PT := "PLCMemory".Offset_Timers.Trilgoten_Stop_Offset);
   "Tag_9" := "Uitlooptimer_Trilgoten".Q;
END_REGION

REGION Network 7: Trilgoten (4) - Reset Drive
   // Reset van Drive Trilgoten (Drive 2)
   RUNG wire#powerrail
      Contact( "Tag_9" )
      R_Coil( "Drive_2_Auto" )
   END_RUNG
   // the same network as SCL:
   IF "Tag_9" THEN "Drive_2_Auto" := FALSE; END_IF;
END_REGION

REGION Network 8: Aanvoerwals (1) - Set Timing as Drive 1
   RUNG wire#powerrail
      Contact( "PLCMemory".TimingSettingOvername )
      Coil( "Overname_Linked_Drive1" )
   END_RUNG
   // the same network as SCL:
   "Overname_Linked_Drive1" := "PLCMemory".TimingSettingOvername;
END_REGION

REGION Network 9: Aanvoerwals (2) - Run Drive (linked to drive 1)
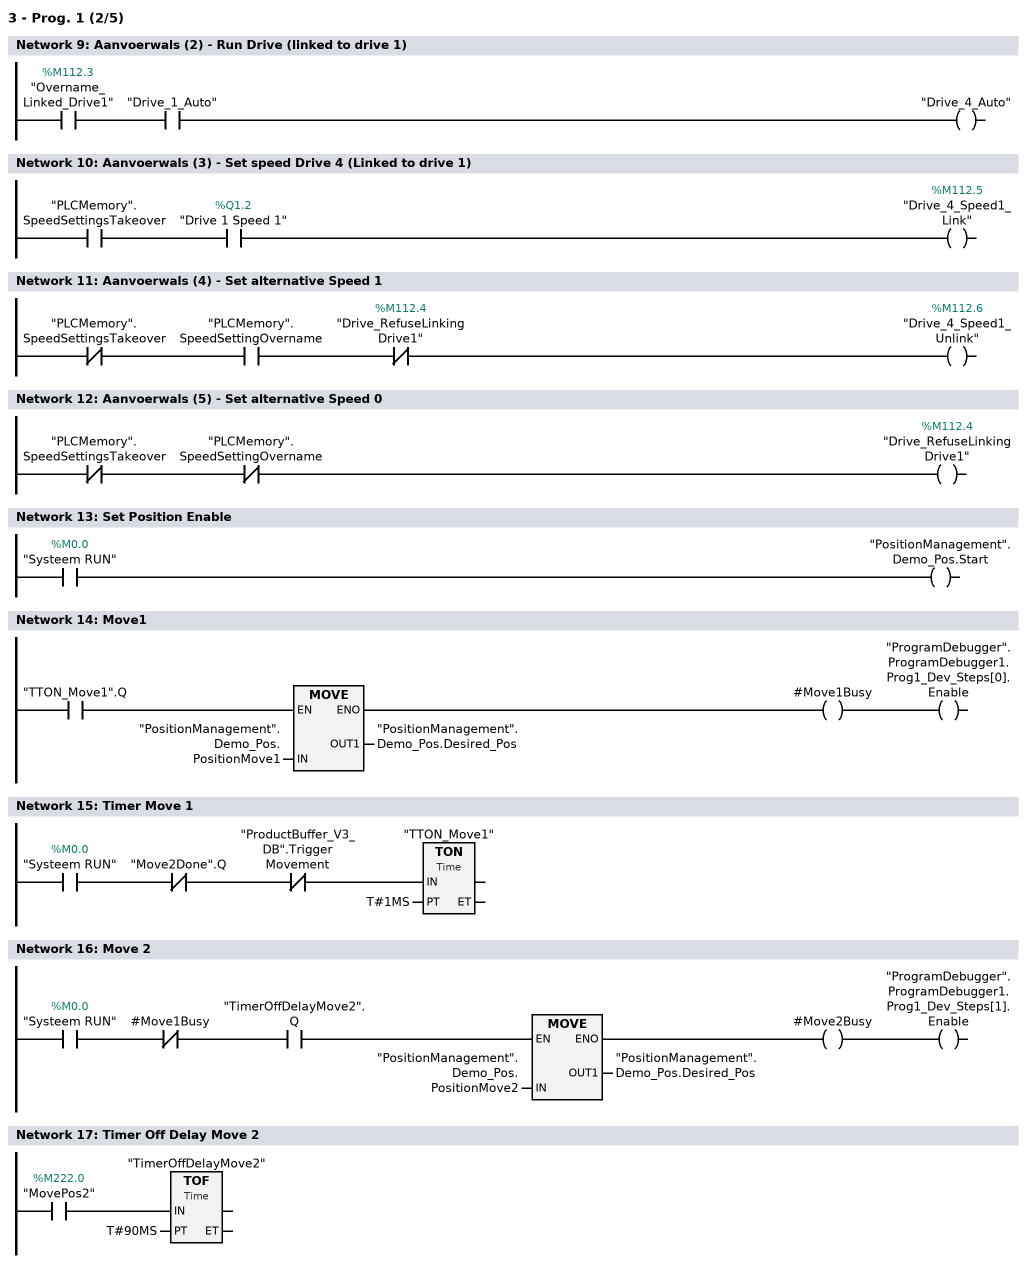
   RUNG wire#powerrail
      Contact( "Overname_Linked_Drive1" )
      Contact( "Drive_1_Auto" )
      Coil( "Drive_4_Auto" )
   END_RUNG
   // the same network as SCL:
   "Drive_4_Auto" := "Overname_Linked_Drive1" AND "Drive_1_Auto";
END_REGION

REGION Network 10: Aanvoerwals (3) - Set speed Drive 4 (Linked to drive 1)
   RUNG wire#powerrail
      Contact( "PLCMemory".SpeedSettingsTakeover )
      Contact( "Drive 1 Speed 1" )
      Coil( "Drive_4_Speed1_Link" )
   END_RUNG
   // the same network as SCL:
   "Drive_4_Speed1_Link" := "PLCMemory".SpeedSettingsTakeover AND "Drive 1 Speed 1";
END_REGION

REGION Network 11: Aanvoerwals (4) - Set alternative Speed 1
   RUNG wire#powerrail
      I_Contact( "PLCMemory".SpeedSettingsTakeover )
      Contact( "PLCMemory".SpeedSettingOvername )
      I_Contact( "Drive_RefuseLinkingDrive1" )
      Coil( "Drive_4_Speed1_Unlink" )
   END_RUNG
   // the same network as SCL:
   "Drive_4_Speed1_Unlink" := NOT "PLCMemory".SpeedSettingsTakeover AND "PLCMemory".SpeedSettingOvername AND NOT "Drive_RefuseLinkingDrive1";
END_REGION

REGION Network 12: Aanvoerwals (5) - Set alternative Speed 0
   RUNG wire#powerrail
      I_Contact( "PLCMemory".SpeedSettingsTakeover )
      I_Contact( "PLCMemory".SpeedSettingOvername )
      Coil( "Drive_RefuseLinkingDrive1" )
   END_RUNG
   // the same network as SCL:
   "Drive_RefuseLinkingDrive1" := NOT "PLCMemory".SpeedSettingsTakeover AND NOT "PLCMemory".SpeedSettingOvername;
END_REGION

REGION Network 13: Set Position Enable
   RUNG wire#powerrail
      Contact( "Systeem RUN" )
      Coil( "PositionManagement".Demo_Pos.Start )
   END_RUNG
   // the same network as SCL:
   "PositionManagement".Demo_Pos.Start := "Systeem RUN";
END_REGION

REGION Network 14: Move1
   RUNG wire#powerrail
      Contact( "TTON_Move1".Q )
      { S7_GenerateENO := "TRUE" } Move(in := "PositionManagement".Demo_Pos.PositionMove1, out1 => "PositionManagement".Demo_Pos.Desired_Pos)
      Coil( #Move1Busy )
      Coil( "ProgramDebugger".ProgramDebugger1.Prog1_Dev_Steps[0].Enable )
   END_RUNG
   // the same network as SCL:
   // ENO of a box is taken as its EN; it also drops when the box reports an error
   IF "TTON_Move1".Q THEN
       "PositionManagement".Demo_Pos.Desired_Pos := "PositionManagement".Demo_Pos.PositionMove1;
   END_IF;
   #Move1Busy := "TTON_Move1".Q;
   "ProgramDebugger".ProgramDebugger1.Prog1_Dev_Steps[0].Enable := "TTON_Move1".Q;
END_REGION

REGION Network 15: Timer Move 1
   RUNG wire#powerrail
      Contact( "Systeem RUN" )
      I_Contact( "Move2Done".Q )
      I_Contact( "ProductBuffer_V3_DB".TriggerMovement )
      { S7_Templates := "time_type := Time" } "TTON_Move1".TON(pt := T#1MS, et =>)
   END_RUNG
   // the same network as SCL:
   "TTON_Move1".TON(IN := "Systeem RUN" AND NOT "Move2Done".Q AND NOT "ProductBuffer_V3_DB".TriggerMovement,
                    PT := T#1MS);
END_REGION

REGION Network 16: Move 2
   RUNG wire#powerrail
      Contact( "Systeem RUN" )
      I_Contact( #Move1Busy )
      Contact( "TimerOffDelayMove2".Q )
      { S7_GenerateENO := "TRUE" } Move(in := "PositionManagement".Demo_Pos.PositionMove2, out1 => "PositionManagement".Demo_Pos.Desired_Pos)
      Coil( #Move2Busy )
      Coil( "ProgramDebugger".ProgramDebugger1.Prog1_Dev_Steps[1].Enable )
   END_RUNG
   // the same network as SCL:
   // ENO of a box is taken as its EN; it also drops when the box reports an error
   #_w1 := "Systeem RUN" AND NOT #Move1Busy AND "TimerOffDelayMove2".Q;
   IF #_w1 THEN
       "PositionManagement".Demo_Pos.Desired_Pos := "PositionManagement".Demo_Pos.PositionMove2;
   END_IF;
   #Move2Busy := #_w1;
   "ProgramDebugger".ProgramDebugger1.Prog1_Dev_Steps[1].Enable := #_w1;
END_REGION

REGION Network 17: Timer Off Delay Move 2
   RUNG wire#powerrail
      Contact( "MovePos2" )
      { S7_Templates := "time_type := Time" } "TimerOffDelayMove2".TOF(pt := T#90MS, et =>)
   END_RUNG
   // the same network as SCL:
   "TimerOffDelayMove2".TOF(IN := "MovePos2", PT := T#90MS);
END_REGION

REGION Network 18: Move2 Done
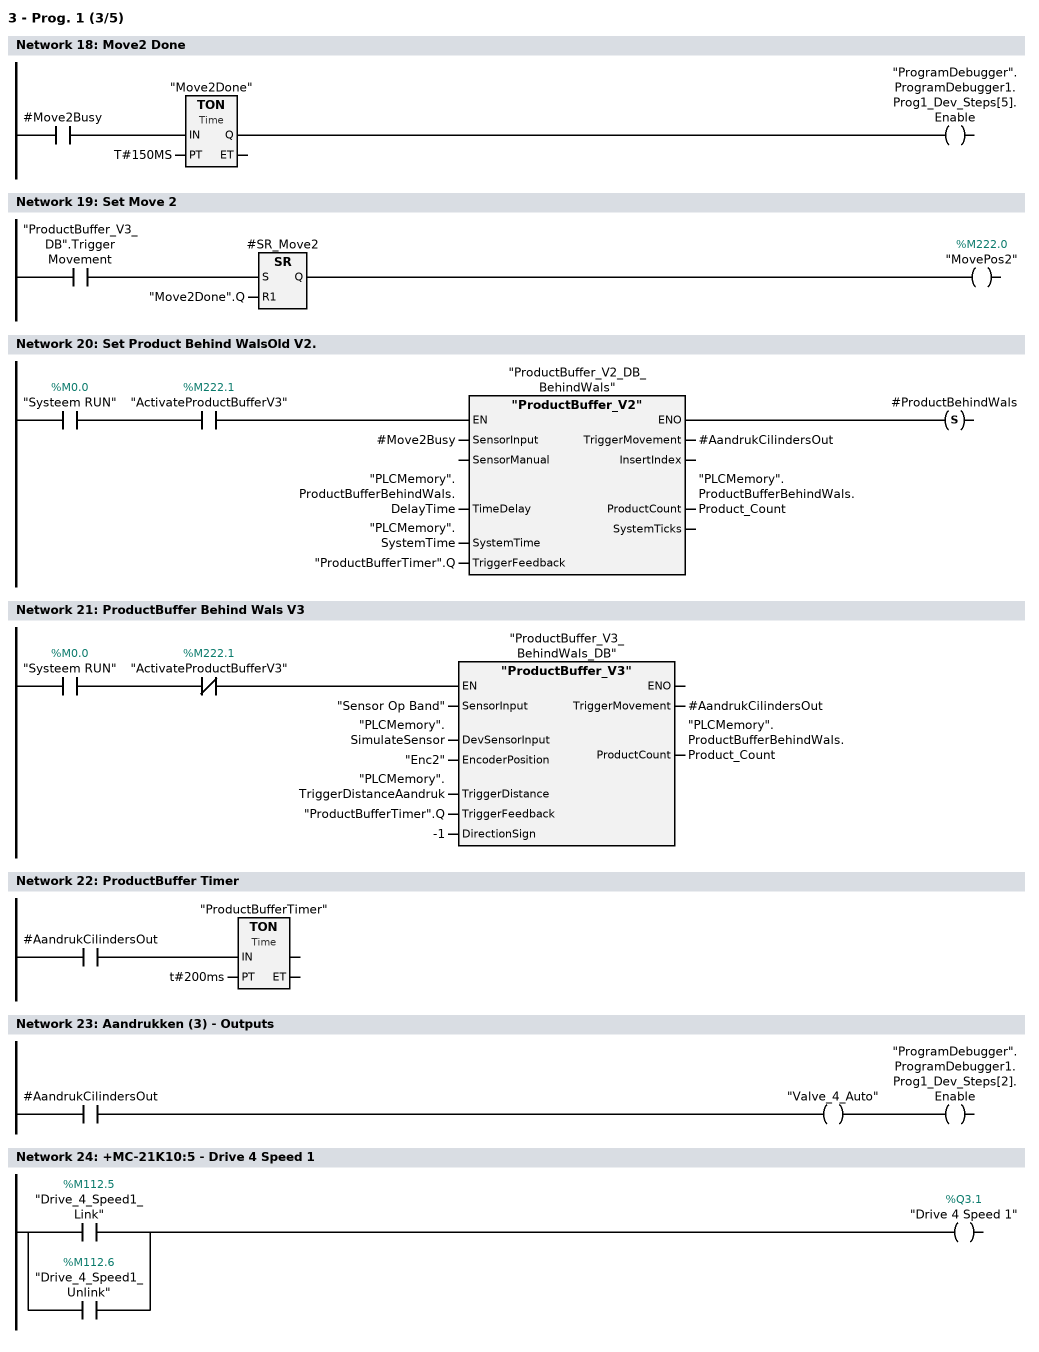
   RUNG wire#powerrail
      Contact( #Move2Busy )
      { S7_Templates := "time_type := Time" } "Move2Done".TON(pt := T#150MS, et =>)
      Coil( "ProgramDebugger".ProgramDebugger1.Prog1_Dev_Steps[5].Enable )
   END_RUNG
   // the same network as SCL:
   "Move2Done".TON(IN := #Move2Busy, PT := T#150MS);
   "ProgramDebugger".ProgramDebugger1.Prog1_Dev_Steps[5].Enable := "Move2Done".Q;
END_REGION

REGION Network 19: Set Move 2
   RUNG wire#powerrail
      Contact( "ProductBuffer_V3_DB".TriggerMovement )
      S_SR(operand := #SR_Move2, r1 := "Move2Done".Q)
      Coil( "MovePos2" )
   END_RUNG
   // the same network as SCL:
   IF "ProductBuffer_V3_DB".TriggerMovement THEN
       #SR_Move2 := TRUE;   // SR flip-flop
   END_IF;
   IF "Move2Done".Q THEN #SR_Move2 := FALSE; END_IF;
   "MovePos2" := #SR_Move2;
END_REGION

REGION Network 20: Set Product Behind WalsOld V2.
   RUNG wire#powerrail
      Contact( "Systeem RUN" )
      Contact( "ActivateProductBufferV3" )
      "ProductBuffer_V2_DB_BehindWals"(SensorInput := #Move2Busy, SensorManual :=, TimeDelay := "PLCMemory".ProductBufferBehindWals.DelayTime, SystemTime := "PLCMemory".SystemTime, TriggerFeedback := "ProductBufferTimer".Q, TriggerMovement => #AandrukCilindersOut, InsertIndex =>, ProductCount => "PLCMemory".ProductBufferBehindWals.Product_Count, SystemTicks =>)
      S_Coil( #ProductBehindWals )
   END_RUNG
   // the same network as SCL:
   "ProductBuffer_V2_DB_BehindWals"(EN := "Systeem RUN" AND "ActivateProductBufferV3",   // "ProductBuffer_V2"
                           SensorInput := #Move2Busy,
                           TimeDelay := "PLCMemory".ProductBufferBehindWals.DelayTime,
                           SystemTime := "PLCMemory".SystemTime,
                           TriggerFeedback := "ProductBufferTimer".Q,
                           TriggerMovement => #AandrukCilindersOut,
                           ProductCount => "PLCMemory".ProductBufferBehindWals.Product_Count,
                           ENO => #_w1);
   IF #_w1 THEN #ProductBehindWals := TRUE; END_IF;
END_REGION

REGION Network 21: ProductBuffer Behind Wals V3
   RUNG wire#powerrail
      Contact( "Systeem RUN" )
      I_Contact( "ActivateProductBufferV3" )
      "ProductBuffer_V3_BehindWals_DB"(SensorInput := "Sensor Op Band", DevSensorInput := "PLCMemory".SimulateSensor, EncoderPosition := "Enc2", TriggerDistance := "PLCMemory".TriggerDistanceAandruk, TriggerFeedback := "ProductBufferTimer".Q, DirectionSign := -1, TriggerMovement => #AandrukCilindersOut, ProductCount => "PLCMemory".ProductBufferBehindWals.Product_Count)
   END_RUNG
   // the same network as SCL:
   IF "Systeem RUN" AND NOT "ActivateProductBufferV3" THEN
       "ProductBuffer_V3_BehindWals_DB"(SensorInput := "Sensor Op Band",   // "ProductBuffer_V3"
                               DevSensorInput := "PLCMemory".SimulateSensor,
                               EncoderPosition := "Enc2",
                               TriggerDistance := "PLCMemory".TriggerDistanceAandruk,
                               TriggerFeedback := "ProductBufferTimer".Q,
                               DirectionSign := -1,
                               TriggerMovement => #AandrukCilindersOut,
                               ProductCount => "PLCMemory".ProductBufferBehindWals.Product_Count);
   END_IF;
END_REGION

REGION Network 22: ProductBuffer Timer
   RUNG wire#powerrail
      Contact( #AandrukCilindersOut )
      { S7_Templates := "time_type := Time" } "ProductBufferTimer".TON(pt := t#200ms, et =>)
   END_RUNG
   // the same network as SCL:
   "ProductBufferTimer".TON(IN := #AandrukCilindersOut, PT := t#200ms);
END_REGION

REGION Network 23: Aandrukken (3) - Outputs
   RUNG wire#powerrail
      Contact( #AandrukCilindersOut )
      Coil( "Valve_4_Auto" )
      Coil( "ProgramDebugger".ProgramDebugger1.Prog1_Dev_Steps[2].Enable )
   END_RUNG
   // the same network as SCL:
   "Valve_4_Auto" := #AandrukCilindersOut;
   "ProgramDebugger".ProgramDebugger1.Prog1_Dev_Steps[2].Enable := #AandrukCilindersOut;
END_REGION

REGION Network 24: +MC-21K10:5 - Drive 4 Speed 1
   RUNG wire#powerrail
      Contact( "Drive_4_Speed1_Link" )
      wire#w1
      Coil( "Drive 4 Speed 1" )
   END_RUNG
   RUNG wire#powerrail
      Contact( "Drive_4_Speed1_Unlink" )
   END_RUNG wire#w1
   // the same network as SCL:
   "Drive 4 Speed 1" := "Drive_4_Speed1_Link" OR "Drive_4_Speed1_Unlink";
END_REGION

REGION Network 25: Retourband (1) - Starttimer
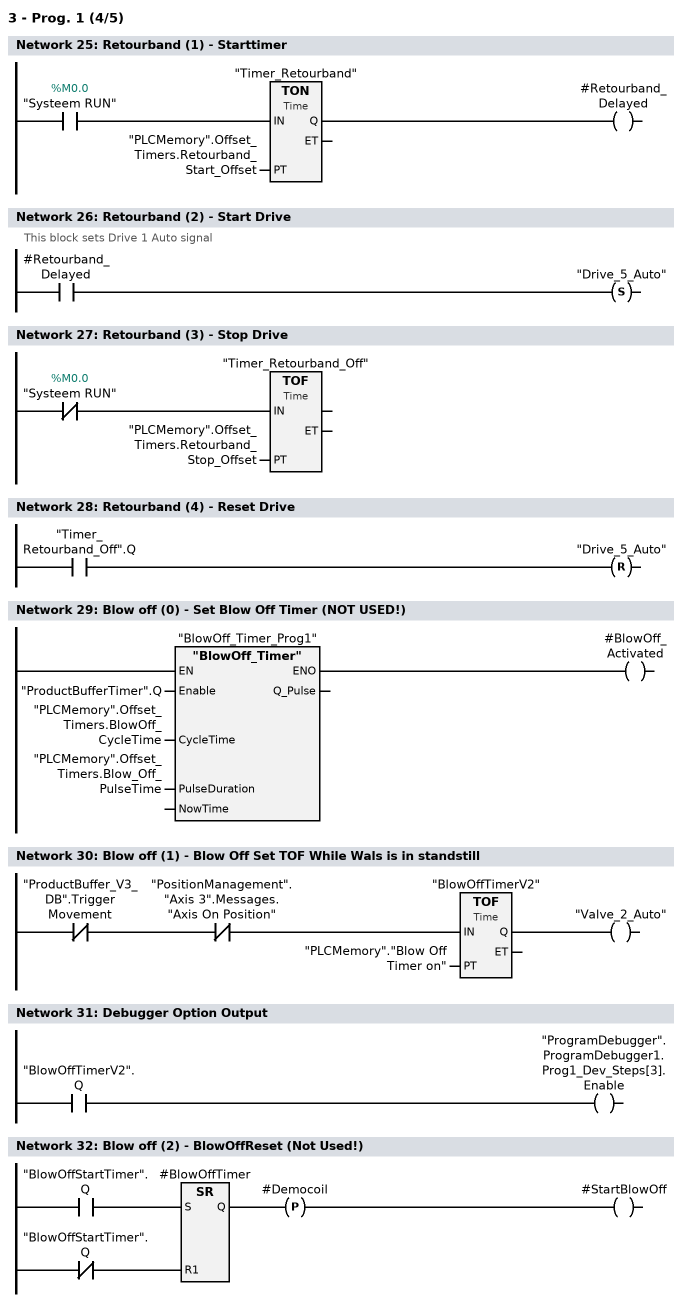
   RUNG wire#powerrail
      Contact( "Systeem RUN" )
      { S7_Templates := "time_type := Time" } "Timer_Retourband".TON(pt := "PLCMemory".Offset_Timers.Retourband_Start_Offset, et =>)
      Coil( #Retourband_Delayed )
   END_RUNG
   // the same network as SCL:
   "Timer_Retourband".TON(IN := "Systeem RUN", PT := "PLCMemory".Offset_Timers.Retourband_Start_Offset);
   #Retourband_Delayed := "Timer_Retourband".Q;
END_REGION

REGION Network 26: Retourband (2) - Start Drive
   // This block sets Drive 1 Auto signal
   RUNG wire#powerrail
      Contact( #Retourband_Delayed )
      S_Coil( "Drive_5_Auto" )
   END_RUNG
   // the same network as SCL:
   IF #Retourband_Delayed THEN "Drive_5_Auto" := TRUE; END_IF;
END_REGION

REGION Network 27: Retourband (3) - Stop Drive
   RUNG wire#powerrail
      I_Contact( "Systeem RUN" )
      { S7_Templates := "time_type := Time" } "Timer_Retourband_Off".TOF(pt := "PLCMemory".Offset_Timers.Retourband_Stop_Offset, et =>)
   END_RUNG
   // the same network as SCL:
   "Timer_Retourband_Off".TOF(IN := NOT "Systeem RUN", PT := "PLCMemory".Offset_Timers.Retourband_Stop_Offset);
END_REGION

REGION Network 28: Retourband (4) - Reset Drive
   RUNG wire#powerrail
      Contact( "Timer_Retourband_Off".Q )
      R_Coil( "Drive_5_Auto" )
   END_RUNG
   // the same network as SCL:
   IF "Timer_Retourband_Off".Q THEN "Drive_5_Auto" := FALSE; END_IF;
END_REGION

REGION Network 29: Blow off (0) - Set Blow Off Timer (NOT USED!)
   RUNG wire#powerrail
      "BlowOff_Timer_Prog1"(Enable := "ProductBufferTimer".Q, CycleTime := "PLCMemory".Offset_Timers.BlowOff_CycleTime, PulseDuration := "PLCMemory".Offset_Timers.Blow_Off_PulseTime, NowTime :=, Q_Pulse =>)
      Coil( #BlowOff_Activated )
   END_RUNG
   // the same network as SCL:
   "BlowOff_Timer_Prog1"(Enable := "ProductBufferTimer".Q,   // "BlowOff_Timer"
                         CycleTime := "PLCMemory".Offset_Timers.BlowOff_CycleTime,
                         PulseDuration := "PLCMemory".Offset_Timers.Blow_Off_PulseTime,
                         ENO => #_w1);
   #BlowOff_Activated := #_w1;
END_REGION

REGION Network 30: Blow off (1) - Blow Off Set TOF While Wals is in standstill
   RUNG wire#powerrail
      I_Contact( "ProductBuffer_V3_DB".TriggerMovement )
      I_Contact( "PositionManagement"."Axis 3".Messages."Axis On Position" )
      { S7_Templates := "time_type := Time" } "BlowOffTimerV2".TOF(pt := "PLCMemory"."Blow Off Timer on", et =>)
      Coil( "Valve_2_Auto" )
   END_RUNG
   // the same network as SCL:
   "BlowOffTimerV2".TOF(IN := NOT "ProductBuffer_V3_DB".TriggerMovement AND NOT "PositionManagement"."Axis 3".Messages."Axis On Position",
                        PT := "PLCMemory"."Blow Off Timer on");
   "Valve_2_Auto" := "BlowOffTimerV2".Q;
END_REGION

REGION Network 31: Debugger Option Output
   RUNG wire#powerrail
      Contact( "BlowOffTimerV2".Q )
      Coil( "ProgramDebugger".ProgramDebugger1.Prog1_Dev_Steps[3].Enable )
   END_RUNG
   // the same network as SCL:
   "ProgramDebugger".ProgramDebugger1.Prog1_Dev_Steps[3].Enable := "BlowOffTimerV2".Q;
END_REGION

REGION Network 32: Blow off (2) - BlowOffReset (Not Used!)
   RUNG wire#powerrail
      Contact( "BlowOffStartTimer".Q )
      S_SR(operand := #BlowOffTimer, r1 := wire#w1)
      P_Trig( #Democoil )
      Coil( #StartBlowOff )
   END_RUNG
   RUNG wire#powerrail
      I_Contact( "BlowOffStartTimer".Q )
   END_RUNG wire#w1
   // the same network as SCL:
   IF "BlowOffStartTimer".Q THEN
       #BlowOffTimer := TRUE;   // SR flip-flop
   END_IF;
   IF NOT "BlowOffStartTimer".Q THEN #BlowOffTimer := FALSE; END_IF;
   #_w1 := #BlowOffTimer AND NOT #Democoil;   // rising edge
   #Democoil := #BlowOffTimer;
   #StartBlowOff := #_w1;
END_REGION

REGION Network 33: PorductBuffer NutStopper
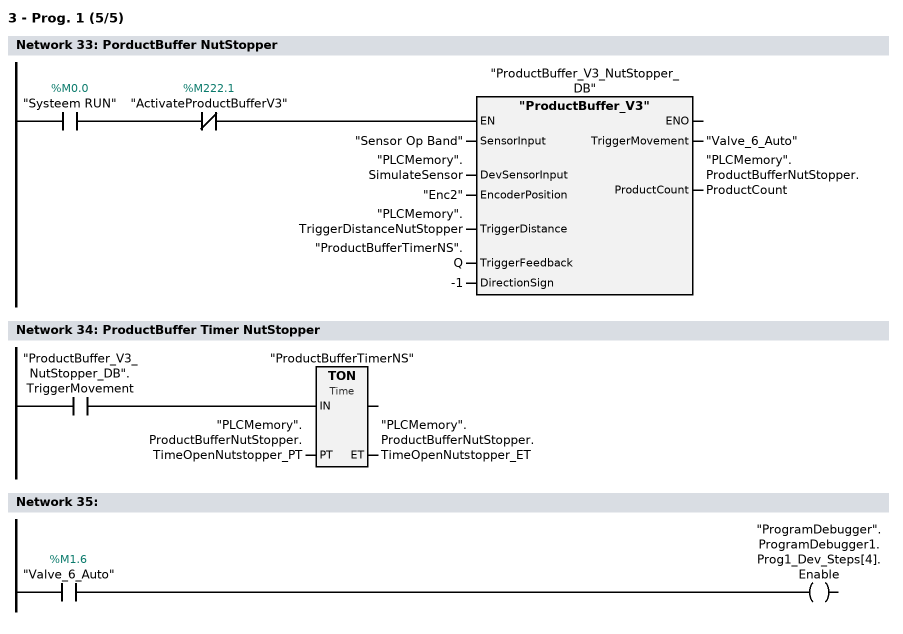
   RUNG wire#powerrail
      Contact( "Systeem RUN" )
      I_Contact( "ActivateProductBufferV3" )
      "ProductBuffer_V3_NutStopper_DB"(SensorInput := "Sensor Op Band", DevSensorInput := "PLCMemory".SimulateSensor, EncoderPosition := "Enc2", TriggerDistance := "PLCMemory".TriggerDistanceNutStopper, TriggerFeedback := "ProductBufferTimerNS".Q, DirectionSign := -1, TriggerMovement => "Valve_6_Auto", ProductCount => "PLCMemory".ProductBufferNutStopper.ProductCount)
   END_RUNG
   // the same network as SCL:
   IF "Systeem RUN" AND NOT "ActivateProductBufferV3" THEN
       "ProductBuffer_V3_NutStopper_DB"(SensorInput := "Sensor Op Band",   // "ProductBuffer_V3"
                               DevSensorInput := "PLCMemory".SimulateSensor,
                               EncoderPosition := "Enc2",
                               TriggerDistance := "PLCMemory".TriggerDistanceNutStopper,
                               TriggerFeedback := "ProductBufferTimerNS".Q,
                               DirectionSign := -1,
                               TriggerMovement => "Valve_6_Auto",
                               ProductCount => "PLCMemory".ProductBufferNutStopper.ProductCount);
   END_IF;
END_REGION

REGION Network 34: ProductBuffer Timer NutStopper
   RUNG wire#powerrail
      Contact( "ProductBuffer_V3_NutStopper_DB".TriggerMovement )
      { S7_Templates := "time_type := Time" } "ProductBufferTimerNS".TON(pt := "PLCMemory".ProductBufferNutStopper.TimeOpenNutstopper_PT, et => "PLCMemory".ProductBufferNutStopper.TimeOpenNutstopper_ET)
   END_RUNG
   // the same network as SCL:
   "ProductBufferTimerNS".TON(IN := "ProductBuffer_V3_NutStopper_DB".TriggerMovement,
                           PT := "PLCMemory".ProductBufferNutStopper.TimeOpenNutstopper_PT,
                           ET => "PLCMemory".ProductBufferNutStopper.TimeOpenNutstopper_ET);
END_REGION

REGION Network 35
   RUNG wire#powerrail
      Contact( "Valve_6_Auto" )
      Coil( "ProgramDebugger".ProgramDebugger1.Prog1_Dev_Steps[4].Enable )
   END_RUNG
   // the same network as SCL:
   "ProgramDebugger".ProgramDebugger1.Prog1_Dev_Steps[4].Enable := "Valve_6_Auto";
END_REGION
END_FUNCTION

FUNCTION_BLOCK "ProductBuffer_V2"
{ S7_Optimized_Access := 'FALSE' }
VERSION : 0.1
   VAR_INPUT 
      SensorInput : Bool;
      SensorManual : Bool;
      TimeDelay : Time;
      SystemTime : Time;
      TriggerFeedback : Bool;
   END_VAR

   VAR_OUTPUT 
      TriggerMovement : Bool;
      InsertIndex { ExternalVisible := 'False'; ExternalWritable := 'False'} : Int;
      ProductCount : Int;
      SystemTicks : DInt;
   END_VAR

   VAR 
      ProductQueue { S7_SetPoint := 'False'} : Array[0..1] of "ProductEntry";
      StartTimes : Struct
         _0 : Time;
         _1 : Time;
         _2 : Time;
         _3 : Time;
         _4 : Time;
         _5 : Time;
         _6 : Time;
         _7 : Time;
         _8 : Time;
         _9 : Time;
      END_STRUCT;
      Actives : Struct
         _0 : Bool;
         _1 : Bool;
         _2 : Bool;
         _3 : Bool;
         _4 : Bool;
         _5 : Bool;
         _6 : Bool;
         _7 : Bool;
         _8 : Bool;
         _9 : Bool;
      END_STRUCT;
      PrevSensor { ExternalVisible := 'False'; ExternalWritable := 'False'} : Bool;
      MovementActive { ExternalVisible := 'False'; ExternalWritable := 'False'} : Bool;
      i { ExternalVisible := 'False'; ExternalWritable := 'False'} : Int;
      Elapsed { ExternalVisible := 'False'; ExternalWritable := 'False'} : DInt;
   END_VAR


BEGIN
	// Flankdetectie sensor
	IF #SensorInput AND NOT #PrevSensor THEN
	    CASE #InsertIndex MOD 10 OF
	        0:
	            IF NOT #Actives._0 THEN
	                #Actives._0 := TRUE;
	                #StartTimes._0 := #SystemTime;
	            END_IF;
	        1:
	            IF NOT #Actives._1 THEN
	                #Actives._1 := TRUE;
	                #StartTimes._1 := #SystemTime;
	            END_IF;
	        2:
	            IF NOT #Actives._2 THEN
	                #Actives._2 := TRUE;
	                #StartTimes._2 := #SystemTime;
	            END_IF;
	        3:
	            IF NOT #Actives._3 THEN
	                #Actives._3 := TRUE;
	                #StartTimes._3 := #SystemTime;
	            END_IF;
	        4:
	            IF NOT #Actives._4 THEN
	                #Actives._4 := TRUE;
	                #StartTimes._4 := #SystemTime;
	            END_IF;
	        5:
	            IF NOT #Actives._5 THEN
	                #Actives._5 := TRUE;
	                #StartTimes._5 := #SystemTime;
	            END_IF;
	        6:
	            IF NOT #Actives._6 THEN
	                #Actives._6 := TRUE;
	                #StartTimes._6 := #SystemTime;
	            END_IF;
	        7:
	            IF NOT #Actives._7 THEN
	                #Actives._7 := TRUE;
	                #StartTimes._7 := #SystemTime;
	            END_IF;
	        8:
	            IF NOT #Actives._8 THEN
	                #Actives._8 := TRUE;
	                #StartTimes._8 := #SystemTime;
	            END_IF;
	        9:
	            IF NOT #Actives._9 THEN
	                #Actives._9 := TRUE;
	                #StartTimes._9 := #SystemTime;
	            END_IF;
	    END_CASE;
	    #InsertIndex := (#InsertIndex + 1) MOD 10;
	END_IF;
	
	#PrevSensor := #SensorInput;
	
	// Tellen hoeveel producten actief zijn
	#ProductCount := 0;
	IF #Actives._0 THEN
	    #ProductCount := #ProductCount + 1;
	END_IF;
	IF #Actives._1 THEN
	    #ProductCount := #ProductCount + 1;
	END_IF;
	IF #Actives._2 THEN
	    #ProductCount := #ProductCount + 1;
	END_IF;
	IF #Actives._3 THEN
	    #ProductCount := #ProductCount + 1;
	END_IF;
	IF #Actives._4 THEN
	    #ProductCount := #ProductCount + 1;
	END_IF;
	IF #Actives._5 THEN
	    #ProductCount := #ProductCount + 1;
	END_IF;
	IF #Actives._6 THEN
	    #ProductCount := #ProductCount + 1;
	END_IF;
	IF #Actives._7 THEN
	    #ProductCount := #ProductCount + 1;
	END_IF;
	IF #Actives._8 THEN
	    #ProductCount := #ProductCount + 1;
	END_IF;
	IF #Actives._9 THEN
	    #ProductCount := #ProductCount + 1;
	END_IF;
	
	// Beweging starten als een product klaar is en geen andere beweging actief is
	IF NOT #MovementActive THEN
	    IF #Actives._0 THEN
	        #Elapsed := TIME_TO_DINT(#SystemTime) - TIME_TO_DINT(#StartTimes._0);
	        IF #Elapsed >= TIME_TO_DINT(#TimeDelay) THEN
	            #TriggerMovement := TRUE;
	            #MovementActive := TRUE;
	            #Actives._0 := FALSE;
	        END_IF;
	    ELSIF #Actives._1 THEN
	        #Elapsed := TIME_TO_DINT(#SystemTime) - TIME_TO_DINT(#StartTimes._1);
	        IF #Elapsed >= TIME_TO_DINT(#TimeDelay) THEN
	            #TriggerMovement := TRUE;
	            #MovementActive := TRUE;
	            #Actives._1 := FALSE;
	        END_IF;
	    ELSIF #Actives._2 THEN
	        #Elapsed := TIME_TO_DINT(#SystemTime) - TIME_TO_DINT(#StartTimes._2);
	        IF #Elapsed >= TIME_TO_DINT(#TimeDelay) THEN
	            #TriggerMovement := TRUE;
	            #MovementActive := TRUE;
	            #Actives._2 := FALSE;
	        END_IF;
	    ELSIF #Actives._3 THEN
	        #Elapsed := TIME_TO_DINT(#SystemTime) - TIME_TO_DINT(#StartTimes._3);
	        IF #Elapsed >= TIME_TO_DINT(#TimeDelay) THEN
	            #TriggerMovement := TRUE;
	            #MovementActive := TRUE;
	            #Actives._3 := FALSE;
	        END_IF;
	    ELSIF #Actives._4 THEN
	        #Elapsed := TIME_TO_DINT(#SystemTime) - TIME_TO_DINT(#StartTimes._4);
	        IF #Elapsed >= TIME_TO_DINT(#TimeDelay) THEN
	            #TriggerMovement := TRUE;
	            #MovementActive := TRUE;
	            #Actives._4 := FALSE;
	        END_IF;
	    ELSIF #Actives._5 THEN
	        #Elapsed := TIME_TO_DINT(#SystemTime) - TIME_TO_DINT(#StartTimes._5);
	        IF #Elapsed >= TIME_TO_DINT(#TimeDelay) THEN
	            #TriggerMovement := TRUE;
	            #MovementActive := TRUE;
	            #Actives._5 := FALSE;
	        END_IF;
	    ELSIF #Actives._6 THEN
	        #Elapsed := TIME_TO_DINT(#SystemTime) - TIME_TO_DINT(#StartTimes._6);
	        IF #Elapsed >= TIME_TO_DINT(#TimeDelay) THEN
	            #TriggerMovement := TRUE;
	            #MovementActive := TRUE;
	            #Actives._6 := FALSE;
	        END_IF;
	    ELSIF #Actives._7 THEN
	        #Elapsed := TIME_TO_DINT(#SystemTime) - TIME_TO_DINT(#StartTimes._7);
	        IF #Elapsed >= TIME_TO_DINT(#TimeDelay) THEN
	            #TriggerMovement := TRUE;
	            #MovementActive := TRUE;
	            #Actives._7 := FALSE;
	        END_IF;
	    ELSIF #Actives._8 THEN
	        #Elapsed := TIME_TO_DINT(#SystemTime) - TIME_TO_DINT(#StartTimes._8);
	        IF #Elapsed >= TIME_TO_DINT(#TimeDelay) THEN
	            #TriggerMovement := TRUE;
	            #MovementActive := TRUE;
	            #Actives._8 := FALSE;
	        END_IF;
	    ELSIF #Actives._9 THEN
	        #Elapsed := TIME_TO_DINT(#SystemTime) - TIME_TO_DINT(#StartTimes._9);
	        IF #Elapsed >= TIME_TO_DINT(#TimeDelay) THEN
	            #TriggerMovement := TRUE;
	            #MovementActive := TRUE;
	            #Actives._9 := FALSE;
	        END_IF;
	    END_IF;
	END_IF;
	
	// Beweging beëindigen na feedback
	IF #MovementActive AND #TriggerFeedback THEN
	    #TriggerMovement := FALSE;
	    #MovementActive := FALSE;
	END_IF;
	
END_FUNCTION_BLOCK

FUNCTION_BLOCK "ProductBuffer_V3"
{ S7_Optimized_Access := 'FALSE' }
VERSION : 0.1
   VAR_INPUT 
      SensorInput : Bool;   // Sensor aan begin band
      DevSensorInput : Bool;
      EncoderPosition : DInt;   // Koppel aan Encoder Data Instance
      TriggerDistance : DInt;   // Gewenste Afstand Product voor trigger
      TriggerFeedback : Bool;
      DirectionSign : DInt;   // irectionSign = +1 for positive counting encoders, -1 for negative counting encoders
   END_VAR

   VAR_OUTPUT 
      TriggerMovement : Bool;   // Trigger Start Movement
      ProductCount : Int;   // Count products in buffer
   END_VAR

   VAR 
      ProductBuffer { S7_SetPoint := 'False'} : Array[0..20] of "ProductTrack";
      PrevSensor { S7_SetPoint := 'True'} : Bool;
      MovementActive : Bool;
      i : Int;
      Distance : DInt;
   END_VAR

   VAR_TEMP 
      AnySensor : Bool;
   END_VAR


BEGIN
	#AnySensor := #SensorInput OR #DevSensorInput;
	// 1️⃣ Flankdetectie - detecteer nieuw product
	IF #AnySensor AND NOT #PrevSensor THEN
	    FOR #i := 0 TO 20 DO
	        IF NOT #ProductBuffer[#i].Active THEN
	            #ProductBuffer[#i].StartPosition := #EncoderPosition;
	            #ProductBuffer[#i].Active := TRUE;
	            EXIT;
	        END_IF;
	    END_FOR;
	END_IF;
	#PrevSensor := #AnySensor;
	
	// 2️⃣ Tel actieve producten
	#ProductCount := 0;
	FOR #i := 0 TO 12 DO
	    IF #ProductBuffer[#i].Active THEN
	        #ProductCount := #ProductCount + 1;
	    END_IF;
	END_FOR;
	
	// DirectionSign = +1 for positive counting encoders, -1 for negative counting encoders
	// Example for your case (negative encoder): DirectionSign := -1;
	
